screen "Prog_Lav2_1" 1366x768
   TextField "Campo de texto_1" at 49,16 size 194x39; Text 'LAVADORA 2'
   TextField "Campo de texto_2" at 49,80 size 103x23; Text 'ENJUAGUES'
   TextField "Campo de texto_3" at 49,112 size 90x23; Text 'INICIALES'
   TextField "Campo de texto_5" at 49,176 size 113x23; Text 'PRE-LAVADO'
   TextField "Campo de texto_10" at 49,336 size 88x23; Text 'LAVADO 1'
   TextField "Campo de texto_14" at 49,464 size 88x23; Text 'LAVADO 2'
   TextField "Campo de texto_18" at 49,592 size 103x23; Text 'ENJUAGUES'
   TextField "Campo de texto_19" at 49,624 size 74x23; Text 'FINALES'
   TextField "Campo de texto_20" at 49,656 size 137x23; Text 'CENTRIFUGADO'
   TextField "Campo de texto_27" at 193,80 size 94x23; Text 'CANTIDAD'
   TextField "Campo de texto_28" at 193,144 size 134x23; Text 'NIVEL DE AGUA'
   TextField "Campo de texto_29" at 193,112 size 70x23; Text 'TIEMPO'
   TextField "Campo de texto_30" at 193,208 size 134x23; Text 'NIVEL DE AGUA'
   TextField "Campo de texto_32" at 193,240 size 140x23; Text 'AGUA CALIENTE'
   TextField "Campo de texto_34" at 193,304 size 132x23; Text 'TEMPERATURA'
   TextField "Campo de texto_35" at 193,336 size 70x23; Text 'TIEMPO'
   TextField "Campo de texto_36" at 193,368 size 134x23; Text 'NIVEL DE AGUA'
   TextField "Campo de texto_37" at 193,400 size 140x23; Text 'AGUA CALIENTE'
   TextField "Campo de texto_38" at 193,432 size 132x23; Text 'TEMPERATURA'
   TextField "Campo de texto_39" at 193,464 size 70x23; Text 'TIEMPO'
   TextField "Campo de texto_40" at 193,496 size 134x23; Text 'NIVEL DE AGUA'
   TextField "Campo de texto_41" at 193,528 size 140x23; Text 'AGUA CALIENTE'
   TextField "Campo de texto_42" at 193,560 size 132x23; Text 'TEMPERATURA'
   TextField "Campo de texto_43" at 193,592 size 94x23; Text 'CANTIDAD'
   TextField "Campo de texto_44" at 193,624 size 70x23; Text 'TIEMPO'
   TextField "Campo de texto_45" at 193,656 size 70x23; Text 'TIEMPO'
   TextField "Campo de texto_4" at 193,272 size 63x23; Text 'VAPOR'
   TextField "Campo de texto_6" at 193,176 size 70x23; Text 'TIEMPO'
   TextField "Campo de texto_7" at 426,39 size 17x33; Text '9'
   TextField "Campo de texto_8" at 537,39 size 34x33; Text '10'
   TextField "Campo de texto_9" at 657,39 size 34x33; Text '11'
   TextField "Campo de texto_11" at 777,39 size 34x33; Text '12'
   TextField "Campo de texto_12" at 897,39 size 34x33; Text '13'
   TextField "Campo de texto_13" at 1017,39 size 34x33; Text '14'
   TextField "Campo de texto_15" at 1137,39 size 34x33; Text '15'
   TextField "Campo de texto_17" at 778,4 size 159x33; Text 'PROGRAMA'
   Button "Botón_1" at 6,695 size 361x66; TextOff 'ATRAS'
      on Click: ActivateScreen("Prog_Lav2_0", 0)
   Button "Botón_2" at 996,694 size 361x66; TextOff 'SIGUIENTE'
      on Click: ActivateScreen("Prog_Lav3_0", 0)
   Button "Botón_3" at 374,694 size 616x66; TextOff 'PRINCIPAL'
      on Click: ActivateScreen("Principal", 0)
   IOField "Campo ES_1" at 394,656 size 80x24; FormatPattern FF; Unit  M
      ProcessValue <- "Lav2_Prog9_Centr_Tiempo"
   IOField "Campo ES_2" at 394,592 size 80x24; FormatPattern F
      ProcessValue <- "Lav2_Prog9_EnjFin_Cant"
   IOField "Campo ES_3" at 394,624 size 80x24; FormatPattern FF; Unit  M
      ProcessValue <- "Lav2_Prog9_EnjFin_Tiempo"
   IOField "Campo ES_4" at 394,80 size 80x24; FormatPattern F
      ProcessValue <- "Lav2_Prog9_EnjIni_Cant"
   IOField "Campo ES_5" at 394,144 size 80x24; FormatPattern F
      ProcessValue <- "Lav2_Prog9_EnjIni_NivAg"
   IOField "Campo ES_6" at 394,112 size 80x24; FormatPattern FF; Unit  M
      ProcessValue <- "Lav2_Prog9_EnjIni_Tiempo"
   IOField "Campo ES_7" at 394,400 size 80x24; FormatPattern F
      ProcessValue <- "Lav2_Prog9_Lav1_AgCaliente"
   IOField "Campo ES_8" at 394,368 size 80x24; FormatPattern F
      ProcessValue <- "Lav2_Prog9_Lav1_NivAg"
   IOField "Campo ES_9" at 394,432 size 80x24; FormatPattern FF; Unit  °C
      ProcessValue <- "Lav2_Prog9_Lav1_Temperatura"
   IOField "Campo ES_10" at 394,336 size 80x24; FormatPattern FF; Unit  M
      ProcessValue <- "Lav2_Prog9_Lav1_Tiempo"
   IOField "Campo ES_11" at 394,528 size 80x24; FormatPattern F
      ProcessValue <- "Lav2_Prog9_Lav2_AgCaliente"
   IOField "Campo ES_12" at 394,496 size 80x24; FormatPattern F
      ProcessValue <- "Lav2_Prog9_Lav2_NivAg"
   IOField "Campo ES_13" at 394,560 size 80x24; FormatPattern FF; Unit °C
      ProcessValue <- "Lav2_Prog9_Lav2_Temperatura"
   IOField "Campo ES_14" at 394,464 size 80x24; FormatPattern FF; Unit  M
      ProcessValue <- "Lav2_Prog9_Lav2_Tiempo"
   IOField "Campo ES_15" at 394,240 size 80x24; FormatPattern F
      ProcessValue <- "Lav2_Prog9_PreLav_AgCaliente"
   IOField "Campo ES_16" at 394,208 size 80x24; FormatPattern F
      ProcessValue <- "Lav2_Prog9_PreLav_NivAg"
   IOField "Campo ES_17" at 394,304 size 80x24; FormatPattern FF; Unit  °C
      ProcessValue <- "Lav2_Prog9_PreLav_Temperatura"
   IOField "Campo ES_18" at 394,176 size 80x24; FormatPattern FF; Unit  M
      ProcessValue <- "Lav2_Prog9_PreLav_Tiempo"
   IOField "Campo ES_19" at 394,272 size 80x24; FormatPattern F
      ProcessValue <- "Lav2_Prog9_PreLav_Vapor"
   IOField "Campo ES_20" at 514,656 size 80x24; FormatPattern FF; Unit  M
      ProcessValue <- "Lav2_Prog10_Centr_Tiempo"
   IOField "Campo ES_21" at 514,592 size 80x24; FormatPattern F
      ProcessValue <- "Lav2_Prog10_EnjFin_Cant"
   IOField "Campo ES_22" at 514,624 size 80x24; FormatPattern FF; Unit  M
      ProcessValue <- "Lav2_Prog10_EnjFin_Tiempo"
   IOField "Campo ES_23" at 514,80 size 80x24; FormatPattern F
      ProcessValue <- "Lav2_Prog10_EnjIni_Cant"
   IOField "Campo ES_24" at 514,144 size 80x24; FormatPattern F
      ProcessValue <- "Lav2_Prog10_EnjIni_NivAg"
   IOField "Campo ES_25" at 514,112 size 80x24; FormatPattern FF; Unit  M
      ProcessValue <- "Lav2_Prog10_EnjIni_Tiempo"
   IOField "Campo ES_26" at 514,400 size 80x24; FormatPattern F
      ProcessValue <- "Lav2_Prog10_Lav1_AgCaliente"
   IOField "Campo ES_27" at 514,368 size 80x24; FormatPattern F
      ProcessValue <- "Lav2_Prog10_Lav1_NivAg"
   IOField "Campo ES_28" at 514,432 size 80x24; FormatPattern FF; Unit  °C
      ProcessValue <- "Lav2_Prog10_Lav1_Temperatura"
   IOField "Campo ES_29" at 514,336 size 80x24; FormatPattern FF; Unit  M
      ProcessValue <- "Lav2_Prog10_Lav1_Tiempo"
   IOField "Campo ES_30" at 514,528 size 80x24; FormatPattern F
      ProcessValue <- "Lav2_Prog10_Lav2_AgCaliente"
   IOField "Campo ES_31" at 514,496 size 80x24; FormatPattern F
      ProcessValue <- "Lav2_Prog10_Lav2_NivAg"
   IOField "Campo ES_32" at 514,560 size 80x24; FormatPattern FF; Unit °C
      ProcessValue <- "Lav2_Prog10_Lav2_Temperatura"
   IOField "Campo ES_33" at 514,464 size 80x24; FormatPattern FF; Unit  M
      ProcessValue <- "Lav2_Prog10_Lav2_Tiempo"
   IOField "Campo ES_34" at 514,240 size 80x24; FormatPattern F
      ProcessValue <- "Lav2_Prog10_PreLav_AgCaliente"
   IOField "Campo ES_35" at 514,208 size 80x24; FormatPattern F
      ProcessValue <- "Lav2_Prog10_PreLav_NivAg"
   IOField "Campo ES_36" at 514,304 size 80x24; FormatPattern FF; Unit  °C
      ProcessValue <- "Lav2_Prog10_PreLav_Temperatura"
   IOField "Campo ES_37" at 514,176 size 80x24; FormatPattern FF; Unit  M
      ProcessValue <- "Lav2_Prog10_PreLav_Tiempo"
   IOField "Campo ES_38" at 514,272 size 80x24; FormatPattern F
      ProcessValue <- "Lav2_Prog10_PreLav_Vapor"
   IOField "Campo ES_39" at 634,656 size 80x24; FormatPattern FF; Unit  M
      ProcessValue <- "Lav2_Prog11_Centr_Tiempo"
   IOField "Campo ES_40" at 634,592 size 80x24; FormatPattern F
      ProcessValue <- "Lav2_Prog11_EnjFin_Cant"
   IOField "Campo ES_41" at 634,624 size 80x24; FormatPattern FF; Unit  M
      ProcessValue <- "Lav2_Prog11_EnjFin_Tiempo"
   IOField "Campo ES_42" at 634,80 size 80x24; FormatPattern F
      ProcessValue <- "Lav2_Prog11_EnjIni_Cant"
   IOField "Campo ES_43" at 634,144 size 80x24; FormatPattern F
      ProcessValue <- "Lav2_Prog11_EnjIni_NivAg"
   IOField "Campo ES_44" at 634,112 size 80x24; FormatPattern FF; Unit  M
      ProcessValue <- "Lav2_Prog11_EnjIni_Tiempo"
   IOField "Campo ES_45" at 634,400 size 80x24; FormatPattern F
      ProcessValue <- "Lav2_Prog11_Lav1_AgCaliente"
   IOField "Campo ES_46" at 634,368 size 80x24; FormatPattern F
      ProcessValue <- "Lav2_Prog11_Lav1_NivAg"
   IOField "Campo ES_47" at 634,432 size 80x24; FormatPattern FF; Unit  °C
      ProcessValue <- "Lav2_Prog11_Lav1_Temperatura"
   IOField "Campo ES_48" at 634,336 size 80x24; FormatPattern FF; Unit  M
      ProcessValue <- "Lav2_Prog11_Lav1_Tiempo"
   IOField "Campo ES_49" at 634,528 size 80x24; FormatPattern F
      ProcessValue <- "Lav2_Prog11_Lav2_AgCaliente"
   IOField "Campo ES_50" at 634,496 size 80x24; FormatPattern F
      ProcessValue <- "Lav2_Prog11_Lav2_NivAg"
   IOField "Campo ES_51" at 634,560 size 80x24; FormatPattern FF; Unit °C
      ProcessValue <- "Lav2_Prog11_Lav2_Temperatura"
   IOField "Campo ES_52" at 634,464 size 80x24; FormatPattern FF; Unit  M
      ProcessValue <- "Lav2_Prog11_Lav2_Tiempo"
   IOField "Campo ES_53" at 634,240 size 80x24; FormatPattern F
      ProcessValue <- "Lav2_Prog11_PreLav_AgCaliente"
   IOField "Campo ES_54" at 634,208 size 80x24; FormatPattern F
      ProcessValue <- "Lav2_Prog11_PreLav_NivAg"
   IOField "Campo ES_55" at 634,304 size 80x24; FormatPattern FF; Unit  °C
      ProcessValue <- "Lav2_Prog11_PreLav_Temperatura"
   IOField "Campo ES_56" at 634,176 size 80x24; FormatPattern FF; Unit  M
      ProcessValue <- "Lav2_Prog11_PreLav_Tiempo"
   IOField "Campo ES_57" at 634,272 size 80x24; FormatPattern F
      ProcessValue <- "Lav2_Prog11_PreLav_Vapor"
   IOField "Campo ES_58" at 754,656 size 80x24; FormatPattern FF; Unit  M
      ProcessValue <- "Lav2_Prog12_Centr_Tiempo"
   IOField "Campo ES_59" at 754,592 size 80x24; FormatPattern F
      ProcessValue <- "Lav2_Prog12_EnjFin_Cant"
   IOField "Campo ES_60" at 754,624 size 80x24; FormatPattern FF; Unit  M
      ProcessValue <- "Lav2_Prog12_EnjFin_Tiempo"
   IOField "Campo ES_61" at 754,80 size 80x24; FormatPattern F
      ProcessValue <- "Lav2_Prog12_EnjIni_Cant"
   IOField "Campo ES_62" at 754,144 size 80x24; FormatPattern F
      ProcessValue <- "Lav2_Prog12_EnjIni_NivAg"
   IOField "Campo ES_63" at 754,112 size 80x24; FormatPattern FF; Unit  M
      ProcessValue <- "Lav2_Prog12_EnjIni_Tiempo"
   IOField "Campo ES_64" at 754,400 size 80x24; FormatPattern F
      ProcessValue <- "Lav2_Prog12_Lav1_AgCaliente"
   IOField "Campo ES_65" at 754,368 size 80x24; FormatPattern F
      ProcessValue <- "Lav2_Prog12_Lav1_NivAg"
   IOField "Campo ES_66" at 754,432 size 80x24; FormatPattern FF; Unit  °C
      ProcessValue <- "Lav2_Prog12_Lav1_Temperatura"
   IOField "Campo ES_67" at 754,336 size 80x24; FormatPattern FF; Unit  M
      ProcessValue <- "Lav2_Prog12_Lav1_Tiempo"
   IOField "Campo ES_68" at 754,528 size 80x24; FormatPattern F
      ProcessValue <- "Lav2_Prog12_Lav2_AgCaliente"
   IOField "Campo ES_69" at 754,496 size 80x24; FormatPattern F
      ProcessValue <- "Lav2_Prog12_Lav2_NivAg"
   IOField "Campo ES_70" at 754,560 size 80x24; FormatPattern FF; Unit °C
      ProcessValue <- "Lav2_Prog12_Lav2_Temperatura"
   IOField "Campo ES_71" at 754,464 size 80x24; FormatPattern FF; Unit  M
      ProcessValue <- "Lav2_Prog12_Lav2_Tiempo"
   IOField "Campo ES_72" at 754,240 size 80x24; FormatPattern F
      ProcessValue <- "Lav2_Prog12_PreLav_AgCaliente"
   IOField "Campo ES_73" at 754,208 size 80x24; FormatPattern F
      ProcessValue <- "Lav2_Prog12_PreLav_NivAg"
   IOField "Campo ES_74" at 754,304 size 80x24; FormatPattern FF; Unit  °C
      ProcessValue <- "Lav2_Prog12_PreLav_Temperatura"
   IOField "Campo ES_75" at 754,176 size 80x24; FormatPattern FF; Unit  M
      ProcessValue <- "Lav2_Prog12_PreLav_Tiempo"
   IOField "Campo ES_76" at 754,272 size 80x24; FormatPattern F
      ProcessValue <- "Lav2_Prog12_PreLav_Vapor"
   IOField "Campo ES_77" at 874,656 size 80x24; FormatPattern FF; Unit  M
      ProcessValue <- "Lav2_Prog13_Centr_Tiempo"
   IOField "Campo ES_78" at 874,592 size 80x24; FormatPattern F
      ProcessValue <- "Lav2_Prog13_EnjFin_Cant"
   IOField "Campo ES_79" at 874,624 size 80x24; FormatPattern FF; Unit  M
      ProcessValue <- "Lav2_Prog13_EnjFin_Tiempo"
   IOField "Campo ES_80" at 874,80 size 80x24; FormatPattern F
      ProcessValue <- "Lav2_Prog13_EnjIni_Cant"
   IOField "Campo ES_81" at 874,144 size 80x24; FormatPattern F
      ProcessValue <- "Lav2_Prog13_EnjIni_NivAg"
   IOField "Campo ES_82" at 874,112 size 80x24; FormatPattern FF; Unit  M
      ProcessValue <- "Lav2_Prog13_EnjIni_Tiempo"
   IOField "Campo ES_83" at 874,400 size 80x24; FormatPattern F
      ProcessValue <- "Lav2_Prog13_Lav1_AgCaliente"
   IOField "Campo ES_84" at 874,368 size 80x24; FormatPattern F
      ProcessValue <- "Lav2_Prog13_Lav1_NivAg"
   IOField "Campo ES_85" at 874,432 size 80x24; FormatPattern FF; Unit  °C
      ProcessValue <- "Lav2_Prog13_Lav1_Temperatura"
   IOField "Campo ES_86" at 874,336 size 80x24; FormatPattern FF; Unit  M
      ProcessValue <- "Lav2_Prog13_Lav1_Tiempo"
   IOField "Campo ES_87" at 874,528 size 80x24; FormatPattern F
      ProcessValue <- "Lav2_Prog13_Lav2_AgCaliente"
   IOField "Campo ES_88" at 874,496 size 80x24; FormatPattern F
      ProcessValue <- "Lav2_Prog13_Lav2_NivAg"
   IOField "Campo ES_89" at 874,560 size 80x24; FormatPattern FF; Unit °C
      ProcessValue <- "Lav2_Prog13_Lav2_Temperatura"
   IOField "Campo ES_90" at 874,464 size 80x24; FormatPattern FF; Unit  M
      ProcessValue <- "Lav2_Prog13_Lav2_Tiempo"
   IOField "Campo ES_91" at 874,240 size 80x24; FormatPattern F
      ProcessValue <- "Lav2_Prog13_PreLav_AgCaliente"
   IOField "Campo ES_92" at 874,208 size 80x24; FormatPattern F
      ProcessValue <- "Lav2_Prog13_PreLav_NivAg"
   IOField "Campo ES_93" at 874,304 size 80x24; FormatPattern FF; Unit  °C
      ProcessValue <- "Lav2_Prog13_PreLav_Temperatura"
   IOField "Campo ES_94" at 874,176 size 80x24; FormatPattern FF; Unit  M
      ProcessValue <- "Lav2_Prog13_PreLav_Tiempo"
   IOField "Campo ES_95" at 874,272 size 80x24; FormatPattern F
      ProcessValue <- "Lav2_Prog13_PreLav_Vapor"
   IOField "Campo ES_96" at 994,656 size 80x24; FormatPattern FF; Unit  M
      ProcessValue <- "Lav2_Prog14_Centr_Tiempo"
   IOField "Campo ES_97" at 994,592 size 80x24; FormatPattern F
      ProcessValue <- "Lav2_Prog14_EnjFin_Cant"
   IOField "Campo ES_98" at 994,624 size 80x24; FormatPattern FF; Unit  M
      ProcessValue <- "Lav2_Prog14_EnjFin_Tiempo"
   IOField "Campo ES_99" at 994,80 size 80x24; FormatPattern F
      ProcessValue <- "Lav2_Prog14_EnjIni_Cant"
   IOField "Campo ES_100" at 994,144 size 80x24; FormatPattern F
      ProcessValue <- "Lav2_Prog14_EnjIni_NivAg"
   IOField "Campo ES_101" at 994,112 size 80x24; FormatPattern FF; Unit  M
      ProcessValue <- "Lav2_Prog14_EnjIni_Tiempo"
   IOField "Campo ES_102" at 994,400 size 80x24; FormatPattern F
      ProcessValue <- "Lav2_Prog14_Lav1_AgCaliente"
   IOField "Campo ES_103" at 994,368 size 80x24; FormatPattern F
      ProcessValue <- "Lav2_Prog14_Lav1_NivAg"
   IOField "Campo ES_104" at 994,432 size 80x24; FormatPattern FF; Unit  °C
      ProcessValue <- "Lav2_Prog14_Lav1_Temperatura"
   IOField "Campo ES_105" at 994,336 size 80x24; FormatPattern FF; Unit  M
      ProcessValue <- "Lav2_Prog14_Lav1_Tiempo"
   IOField "Campo ES_106" at 994,528 size 80x24; FormatPattern F
      ProcessValue <- "Lav2_Prog14_Lav2_AgCaliente"
   IOField "Campo ES_107" at 994,496 size 80x24; FormatPattern F
      ProcessValue <- "Lav2_Prog14_Lav2_NivAg"
   IOField "Campo ES_108" at 994,560 size 80x24; FormatPattern FF; Unit °C
      ProcessValue <- "Lav2_Prog14_Lav2_Temperatura"
   IOField "Campo ES_109" at 994,464 size 80x24; FormatPattern FF; Unit  M
      ProcessValue <- "Lav2_Prog14_Lav2_Tiempo"
   IOField "Campo ES_110" at 994,240 size 80x24; FormatPattern F
      ProcessValue <- "Lav2_Prog14_PreLav_AgCaliente"
   IOField "Campo ES_111" at 994,208 size 80x24; FormatPattern F
      ProcessValue <- "Lav2_Prog14_PreLav_NivAg"
   IOField "Campo ES_112" at 994,304 size 80x24; FormatPattern FF; Unit  °C
      ProcessValue <- "Lav2_Prog14_PreLav_Temperatura"
   IOField "Campo ES_113" at 994,176 size 80x24; FormatPattern FF; Unit  M
      ProcessValue <- "Lav2_Prog14_PreLav_Tiempo"
   IOField "Campo ES_114" at 994,272 size 80x24; FormatPattern F
      ProcessValue <- "Lav2_Prog14_PreLav_Vapor"
   IOField "Campo ES_115" at 1114,656 size 80x24; FormatPattern FF; Unit  M
      ProcessValue <- "Lav2_Prog15_Centr_Tiempo"
   IOField "Campo ES_116" at 1114,592 size 80x24; FormatPattern F
      ProcessValue <- "Lav2_Prog15_EnjFin_Cant"
   IOField "Campo ES_117" at 1114,624 size 80x24; FormatPattern FF; Unit  M
      ProcessValue <- "Lav2_Prog15_EnjFin_Tiempo"
   IOField "Campo ES_118" at 1114,80 size 80x24; FormatPattern F
      ProcessValue <- "Lav2_Prog15_EnjIni_Cant"
   IOField "Campo ES_119" at 1114,144 size 80x24; FormatPattern F
      ProcessValue <- "Lav2_Prog15_EnjIni_NivAg"
   IOField "Campo ES_120" at 1114,112 size 80x24; FormatPattern FF; Unit  M
      ProcessValue <- "Lav2_Prog15_EnjIni_Tiempo"
   IOField "Campo ES_121" at 1114,400 size 80x24; FormatPattern F
      ProcessValue <- "Lav2_Prog15_Lav1_AgCaliente"
   IOField "Campo ES_122" at 1114,368 size 80x24; FormatPattern F
      ProcessValue <- "Lav2_Prog15_Lav1_NivAg"
   IOField "Campo ES_123" at 1114,432 size 80x24; FormatPattern FF; Unit  °C
      ProcessValue <- "Lav2_Prog15_Lav1_Temperatura"
   IOField "Campo ES_124" at 1114,336 size 80x24; FormatPattern FF; Unit  M
      ProcessValue <- "Lav2_Prog15_Lav1_Tiempo"
   IOField "Campo ES_125" at 1114,528 size 80x24; FormatPattern F
      ProcessValue <- "Lav2_Prog15_Lav2_AgCaliente"
   IOField "Campo ES_126" at 1114,496 size 80x24; FormatPattern F
      ProcessValue <- "Lav2_Prog15_Lav2_NivAg"
   IOField "Campo ES_127" at 1114,560 size 80x24; FormatPattern FF; Unit °C
      ProcessValue <- "Lav2_Prog15_Lav2_Temperatura"
   IOField "Campo ES_128" at 1114,464 size 80x24; FormatPattern FF; Unit  M
      ProcessValue <- "Lav2_Prog15_Lav2_Tiempo"
   IOField "Campo ES_129" at 1114,240 size 80x24; FormatPattern F
      ProcessValue <- "Lav2_Prog15_PreLav_AgCaliente"
   IOField "Campo ES_130" at 1114,208 size 80x24; FormatPattern F
      ProcessValue <- "Lav2_Prog15_PreLav_NivAg"
   IOField "Campo ES_131" at 1114,304 size 80x24; FormatPattern FF; Unit  °C
      ProcessValue <- "Lav2_Prog15_PreLav_Temperatura"
   IOField "Campo ES_132" at 1114,176 size 80x24; FormatPattern FF; Unit  M
      ProcessValue <- "Lav2_Prog15_PreLav_Tiempo"
   IOField "Campo ES_133" at 1114,272 size 80x24; FormatPattern F
      ProcessValue <- "Lav2_Prog15_PreLav_Vapor"

screen "Prog_Lav3_0" 1366x768
   TextField "Campo de texto_1" at 49,16 size 194x39; Text 'LAVADORA 3'
   TextField "Campo de texto_2" at 49,80 size 103x23; Text 'ENJUAGUES'
   TextField "Campo de texto_3" at 49,112 size 90x23; Text 'INICIALES'
   TextField "Campo de texto_5" at 49,176 size 113x23; Text 'PRE-LAVADO'
   TextField "Campo de texto_10" at 49,336 size 88x23; Text 'LAVADO 1'
   TextField "Campo de texto_14" at 49,464 size 88x23; Text 'LAVADO 2'
   TextField "Campo de texto_18" at 49,592 size 103x23; Text 'ENJUAGUES'
   TextField "Campo de texto_19" at 49,624 size 74x23; Text 'FINALES'
   TextField "Campo de texto_20" at 49,656 size 137x23; Text 'CENTRIFUGADO'
   TextField "Campo de texto_27" at 193,80 size 94x23; Text 'CANTIDAD'
   TextField "Campo de texto_28" at 193,144 size 134x23; Text 'NIVEL DE AGUA'
   TextField "Campo de texto_29" at 193,112 size 70x23; Text 'TIEMPO'
   TextField "Campo de texto_30" at 193,208 size 134x23; Text 'NIVEL DE AGUA'
   TextField "Campo de texto_32" at 193,240 size 140x23; Text 'AGUA CALIENTE'
   TextField "Campo de texto_34" at 193,304 size 132x23; Text 'TEMPERATURA'
   TextField "Campo de texto_35" at 193,336 size 70x23; Text 'TIEMPO'
   TextField "Campo de texto_36" at 193,368 size 134x23; Text 'NIVEL DE AGUA'
   TextField "Campo de texto_37" at 193,400 size 140x23; Text 'AGUA CALIENTE'
   TextField "Campo de texto_38" at 193,432 size 132x23; Text 'TEMPERATURA'
   TextField "Campo de texto_39" at 193,464 size 70x23; Text 'TIEMPO'
   TextField "Campo de texto_40" at 193,496 size 134x23; Text 'NIVEL DE AGUA'
   TextField "Campo de texto_41" at 193,528 size 140x23; Text 'AGUA CALIENTE'
   TextField "Campo de texto_42" at 193,560 size 132x23; Text 'TEMPERATURA'
   TextField "Campo de texto_43" at 193,592 size 94x23; Text 'CANTIDAD'
   TextField "Campo de texto_44" at 193,624 size 70x23; Text 'TIEMPO'
   TextField "Campo de texto_45" at 193,656 size 70x23; Text 'TIEMPO'
   TextField "Campo de texto_4" at 193,272 size 63x23; Text 'VAPOR'
   TextField "Campo de texto_6" at 193,176 size 70x23; Text 'TIEMPO'
   TextField "Campo de texto_7" at 426,39 size 17x33; Text '1'
   TextField "Campo de texto_8" at 546,39 size 17x33; Text '2'
   TextField "Campo de texto_9" at 666,39 size 17x33; Text '3'
   TextField "Campo de texto_11" at 786,39 size 17x33; Text '4'
   TextField "Campo de texto_12" at 906,39 size 17x33; Text '5'
   TextField "Campo de texto_13" at 1026,39 size 17x33; Text '6'
   TextField "Campo de texto_15" at 1146,39 size 17x33; Text '7'
   TextField "Campo de texto_16" at 1266,39 size 17x33; Text '8'
   TextField "Campo de texto_17" at 778,4 size 159x33; Text 'PROGRAMA'
   Button "Botón_1" at 6,695 size 361x66; TextOff 'ATRAS'
      on Click: ActivateScreen("Prog_Lav2_1", 0)
   Button "Botón_2" at 996,694 size 361x66; TextOff 'SIGUIENTE'
      on Click: ActivateScreen("Prog_Lav3_1", 0)
   Button "Botón_3" at 374,694 size 616x66; TextOff 'PRINCIPAL'
      on Click: ActivateScreen("Principal", 0)
   IOField "Campo ES_1" at 394,656 size 80x24; FormatPattern FF; Unit  M
      ProcessValue <- "Lav3_Prog1_Centr_Tiempo"
   IOField "Campo ES_2" at 394,592 size 80x24; FormatPattern F
      ProcessValue <- "Lav3_Prog1_EnjFin_Cant"
   IOField "Campo ES_3" at 394,624 size 80x24; FormatPattern FF; Unit  M
      ProcessValue <- "Lav3_Prog1_EnjFin_Tiempo"
   IOField "Campo ES_4" at 394,80 size 80x24; FormatPattern F
      ProcessValue <- "Lav3_Prog1_EnjIni_Cant"
   IOField "Campo ES_5" at 394,144 size 80x24; FormatPattern F
      ProcessValue <- "Lav3_Prog1_EnjIni_NivAg"
   IOField "Campo ES_6" at 394,112 size 80x24; FormatPattern FF; Unit  M
      ProcessValue <- "Lav3_Prog1_EnjIni_Tiempo"
   IOField "Campo ES_7" at 394,400 size 80x24; FormatPattern F
      ProcessValue <- "Lav3_Prog1_Lav1_AgCaliente"
   IOField "Campo ES_8" at 394,368 size 80x24; FormatPattern F
      ProcessValue <- "Lav3_Prog1_Lav1_NivAg"
   IOField "Campo ES_9" at 394,432 size 80x24; FormatPattern FF; Unit  °C
      ProcessValue <- "Lav3_Prog1_Lav1_Temperatura"
   IOField "Campo ES_10" at 394,336 size 80x24; FormatPattern FF; Unit  M
      ProcessValue <- "Lav3_Prog1_Lav1_Tiempo"
   IOField "Campo ES_11" at 394,528 size 80x24; FormatPattern F
      ProcessValue <- "Lav3_Prog1_Lav2_AgCaliente"
   IOField "Campo ES_12" at 394,496 size 80x24; FormatPattern F
      ProcessValue <- "Lav3_Prog1_Lav2_NivAg"
   IOField "Campo ES_13" at 394,560 size 80x24; FormatPattern FF; Unit °C
      ProcessValue <- "Lav3_Prog1_Lav2_Temperatura"
   IOField "Campo ES_14" at 394,464 size 80x24; FormatPattern FF; Unit  M
      ProcessValue <- "Lav3_Prog1_Lav2_Tiempo"
   IOField "Campo ES_15" at 394,240 size 80x24; FormatPattern F
      ProcessValue <- "Lav3_Prog1_PreLav_AgCaliente"
   IOField "Campo ES_16" at 394,208 size 80x24; FormatPattern F
      ProcessValue <- "Lav3_Prog1_PreLav_NivAg"
   IOField "Campo ES_17" at 394,304 size 80x24; FormatPattern FF; Unit  °C
      ProcessValue <- "Lav3_Prog1_PreLav_Temperatura"
   IOField "Campo ES_18" at 394,176 size 80x24; FormatPattern FF; Unit  M
      ProcessValue <- "Lav3_Prog1_PreLav_Tiempo"
   IOField "Campo ES_19" at 394,272 size 80x24; FormatPattern F
      ProcessValue <- "Lav3_Prog1_PreLav_Vapor"
   IOField "Campo ES_20" at 514,656 size 80x24; FormatPattern FF; Unit  M
      ProcessValue <- "Lav3_Prog2_Centr_Tiempo"
   IOField "Campo ES_21" at 514,592 size 80x24; FormatPattern F
      ProcessValue <- "Lav3_Prog2_EnjFin_Cant"
   IOField "Campo ES_22" at 514,624 size 80x24; FormatPattern FF; Unit  M
      ProcessValue <- "Lav3_Prog2_EnjFin_Tiempo"
   IOField "Campo ES_23" at 514,80 size 80x24; FormatPattern F
      ProcessValue <- "Lav3_Prog2_EnjIni_Cant"
   IOField "Campo ES_24" at 514,144 size 80x24; FormatPattern F
      ProcessValue <- "Lav3_Prog2_EnjIni_NivAg"
   IOField "Campo ES_25" at 514,112 size 80x24; FormatPattern FF; Unit  M
      ProcessValue <- "Lav3_Prog2_EnjIni_Tiempo"
   IOField "Campo ES_26" at 514,400 size 80x24; FormatPattern F
      ProcessValue <- "Lav3_Prog2_Lav1_AgCaliente"
   IOField "Campo ES_27" at 514,368 size 80x24; FormatPattern F
      ProcessValue <- "Lav3_Prog2_Lav1_NivAg"
   IOField "Campo ES_28" at 514,432 size 80x24; FormatPattern FF; Unit  °C
      ProcessValue <- "Lav3_Prog2_Lav1_Temperatura"
   IOField "Campo ES_29" at 514,336 size 80x24; FormatPattern FF; Unit  M
      ProcessValue <- "Lav3_Prog2_Lav1_Tiempo"
   IOField "Campo ES_30" at 514,528 size 80x24; FormatPattern F
      ProcessValue <- "Lav3_Prog2_Lav2_AgCaliente"
   IOField "Campo ES_31" at 514,496 size 80x24; FormatPattern F
      ProcessValue <- "Lav3_Prog2_Lav2_NivAg"
   IOField "Campo ES_32" at 514,560 size 80x24; FormatPattern FF; Unit °C
      ProcessValue <- "Lav3_Prog2_Lav2_Temperatura"
   IOField "Campo ES_33" at 514,464 size 80x24; FormatPattern FF; Unit  M
      ProcessValue <- "Lav3_Prog2_Lav2_Tiempo"
   IOField "Campo ES_34" at 514,240 size 80x24; FormatPattern F
      ProcessValue <- "Lav3_Prog2_PreLav_AgCaliente"
   IOField "Campo ES_35" at 514,208 size 80x24; FormatPattern F
      ProcessValue <- "Lav3_Prog2_PreLav_NivAg"
   IOField "Campo ES_36" at 514,304 size 80x24; FormatPattern FF; Unit  °C
      ProcessValue <- "Lav3_Prog2_PreLav_Temperatura"
   IOField "Campo ES_37" at 514,176 size 80x24; FormatPattern FF; Unit  M
      ProcessValue <- "Lav3_Prog2_PreLav_Tiempo"
   IOField "Campo ES_38" at 514,272 size 80x24; FormatPattern F
      ProcessValue <- "Lav3_Prog2_PreLav_Vapor"
   IOField "Campo ES_39" at 634,656 size 80x24; FormatPattern FF; Unit  M
      ProcessValue <- "Lav3_Prog3_Centr_Tiempo"
   IOField "Campo ES_40" at 634,592 size 80x24; FormatPattern F
      ProcessValue <- "Lav3_Prog3_EnjFin_Cant"
   IOField "Campo ES_41" at 634,624 size 80x24; FormatPattern FF; Unit  M
      ProcessValue <- "Lav3_Prog3_EnjFin_Tiempo"
   IOField "Campo ES_42" at 634,80 size 80x24; FormatPattern F
      ProcessValue <- "Lav3_Prog3_EnjIni_Cant"
   IOField "Campo ES_43" at 634,144 size 80x24; FormatPattern F
      ProcessValue <- "Lav3_Prog3_EnjIni_NivAg"
   IOField "Campo ES_44" at 634,112 size 80x24; FormatPattern FF; Unit  M
      ProcessValue <- "Lav3_Prog3_EnjIni_Tiempo"
   IOField "Campo ES_45" at 634,400 size 80x24; FormatPattern F
      ProcessValue <- "Lav3_Prog3_Lav1_AgCaliente"
   IOField "Campo ES_46" at 634,368 size 80x24; FormatPattern F
      ProcessValue <- "Lav3_Prog3_Lav1_NivAg"
   IOField "Campo ES_47" at 634,432 size 80x24; FormatPattern FF; Unit  °C
      ProcessValue <- "Lav3_Prog3_Lav1_Temperatura"
   IOField "Campo ES_48" at 634,336 size 80x24; FormatPattern FF; Unit  M
      ProcessValue <- "Lav3_Prog3_Lav1_Tiempo"
   IOField "Campo ES_49" at 634,528 size 80x24; FormatPattern F
      ProcessValue <- "Lav3_Prog3_Lav2_AgCaliente"
   IOField "Campo ES_50" at 634,496 size 80x24; FormatPattern F
      ProcessValue <- "Lav3_Prog3_Lav2_NivAg"
   IOField "Campo ES_51" at 634,560 size 80x24; FormatPattern FF; Unit °C
      ProcessValue <- "Lav3_Prog3_Lav2_Temperatura"
   IOField "Campo ES_52" at 634,464 size 80x24; FormatPattern FF; Unit  M
      ProcessValue <- "Lav3_Prog3_Lav2_Tiempo"
   IOField "Campo ES_53" at 634,240 size 80x24; FormatPattern F
      ProcessValue <- "Lav3_Prog3_PreLav_AgCaliente"
   IOField "Campo ES_54" at 634,208 size 80x24; FormatPattern F
      ProcessValue <- "Lav3_Prog3_PreLav_NivAg"
   IOField "Campo ES_55" at 634,304 size 80x24; FormatPattern FF; Unit  °C
      ProcessValue <- "Lav3_Prog3_PreLav_Temperatura"
   IOField "Campo ES_56" at 634,176 size 80x24; FormatPattern FF; Unit  M
      ProcessValue <- "Lav3_Prog3_PreLav_Tiempo"
   IOField "Campo ES_57" at 634,272 size 80x24; FormatPattern F
      ProcessValue <- "Lav3_Prog3_PreLav_Vapor"
   IOField "Campo ES_58" at 754,656 size 80x24; FormatPattern FF; Unit  M
      ProcessValue <- "Lav3_Prog4_Centr_Tiempo"
   IOField "Campo ES_59" at 754,592 size 80x24; FormatPattern F
      ProcessValue <- "Lav1_Prog4_EnjFin_Cant"
   IOField "Campo ES_60" at 754,624 size 80x24; FormatPattern FF; Unit  M
      ProcessValue <- "Lav1_Prog4_EnjFin_Tiempo"
   IOField "Campo ES_61" at 754,80 size 80x24; FormatPattern F
      ProcessValue <- "Lav1_Prog4_EnjIni_Cant"
   IOField "Campo ES_62" at 754,144 size 80x24; FormatPattern F
      ProcessValue <- "Lav1_Prog4_EnjIni_NivAg"
   IOField "Campo ES_63" at 754,112 size 80x24; FormatPattern FF; Unit  M
      ProcessValue <- "Lav1_Prog4_EnjIni_Tiempo"
   IOField "Campo ES_64" at 754,400 size 80x24; FormatPattern F
      ProcessValue <- "Lav1_Prog4_Lav1_AgCaliente"
   IOField "Campo ES_65" at 754,368 size 80x24; FormatPattern F
      ProcessValue <- "Lav1_Prog4_Lav1_NivAg"
   IOField "Campo ES_66" at 754,432 size 80x24; FormatPattern FF; Unit  °C
      ProcessValue <- "Lav1_Prog4_Lav1_Temperatura"
   IOField "Campo ES_67" at 754,336 size 80x24; FormatPattern FF; Unit  M
      ProcessValue <- "Lav1_Prog4_Lav1_Tiempo"
   IOField "Campo ES_68" at 754,528 size 80x24; FormatPattern F
      ProcessValue <- "Lav1_Prog4_Lav2_AgCaliente"
   IOField "Campo ES_69" at 754,496 size 80x24; FormatPattern F
      ProcessValue <- "Lav1_Prog4_Lav2_NivAg"
   IOField "Campo ES_70" at 754,560 size 80x24; FormatPattern FF; Unit °C
      ProcessValue <- "Lav1_Prog4_Lav2_Temperatura"
   IOField "Campo ES_71" at 754,464 size 80x24; FormatPattern FF; Unit  M
      ProcessValue <- "Lav1_Prog4_Lav2_Tiempo"
   IOField "Campo ES_72" at 754,240 size 80x24; FormatPattern F
      ProcessValue <- "Lav1_Prog4_PreLav_AgCaliente"
   IOField "Campo ES_73" at 754,208 size 80x24; FormatPattern F
      ProcessValue <- "Lav1_Prog4_PreLav_NivAg"
   IOField "Campo ES_74" at 754,304 size 80x24; FormatPattern FF; Unit  °C
      ProcessValue <- "Lav1_Prog4_PreLav_Temperatura"
   IOField "Campo ES_75" at 754,176 size 80x24; FormatPattern FF; Unit  M
      ProcessValue <- "Lav1_Prog4_PreLav_Tiempo"
   IOField "Campo ES_76" at 754,272 size 80x24; FormatPattern F
      ProcessValue <- "Lav1_Prog4_PreLav_Vapor"
   IOField "Campo ES_77" at 874,656 size 80x24; FormatPattern FF; Unit  M
      ProcessValue <- "Lav3_Prog6_Centr_Tiempo"
   IOField "Campo ES_78" at 874,592 size 80x24; FormatPattern F
      ProcessValue <- "Lav3_Prog6_EnjFin_Cant"
   IOField "Campo ES_79" at 874,624 size 80x24; FormatPattern FF; Unit  M
      ProcessValue <- "Lav3_Prog6_EnjFin_Tiempo"
   IOField "Campo ES_80" at 874,80 size 80x24; FormatPattern F
      ProcessValue <- "Lav3_Prog5_EnjIni_Cant"
   IOField "Campo ES_81" at 874,144 size 80x24; FormatPattern F
      ProcessValue <- "Lav3_Prog5_EnjIni_NivAg"
   IOField "Campo ES_82" at 874,112 size 80x24; FormatPattern FF; Unit  M
      ProcessValue <- "Lav3_Prog5_EnjIni_Tiempo"
   IOField "Campo ES_83" at 874,400 size 80x24; FormatPattern F
      ProcessValue <- "Lav3_Prog5_Lav1_AgCaliente"
   IOField "Campo ES_84" at 874,368 size 80x24; FormatPattern F
      ProcessValue <- "Lav3_Prog5_Lav1_NivAg"
   IOField "Campo ES_85" at 874,432 size 80x24; FormatPattern FF; Unit  °C
      ProcessValue <- "Lav3_Prog5_Lav1_Temperatura"
   IOField "Campo ES_86" at 874,336 size 80x24; FormatPattern FF; Unit  M
      ProcessValue <- "Lav3_Prog5_Lav1_Tiempo"
   IOField "Campo ES_87" at 874,528 size 80x24; FormatPattern F
      ProcessValue <- "Lav3_Prog6_Lav2_AgCaliente"
   IOField "Campo ES_88" at 874,496 size 80x24; FormatPattern F
      ProcessValue <- "Lav3_Prog6_Lav2_NivAg"
   IOField "Campo ES_89" at 874,560 size 80x24; FormatPattern FF; Unit °C
      ProcessValue <- "Lav3_Prog6_Lav2_Temperatura"
   IOField "Campo ES_90" at 874,464 size 80x24; FormatPattern FF; Unit  M
      ProcessValue <- "Lav3_Prog6_Lav2_Tiempo"
   IOField "Campo ES_91" at 874,240 size 80x24; FormatPattern F
      ProcessValue <- "Lav3_Prog5_PreLav_AgCaliente"
   IOField "Campo ES_92" at 874,208 size 80x24; FormatPattern F
      ProcessValue <- "Lav3_Prog5_PreLav_NivAg"
   IOField "Campo ES_93" at 874,304 size 80x24; FormatPattern FF; Unit  °C
      ProcessValue <- "Lav3_Prog5_PreLav_Temperatura"
   IOField "Campo ES_94" at 874,176 size 80x24; FormatPattern FF; Unit  M
      ProcessValue <- "Lav3_Prog5_PreLav_Tiempo"
   IOField "Campo ES_95" at 874,272 size 80x24; FormatPattern F
      ProcessValue <- "Lav3_Prog5_PreLav_Vapor"
   IOField "Campo ES_96" at 994,656 size 80x24; FormatPattern FF; Unit  M
      ProcessValue <- "Lav3_Prog6_Centr_Tiempo"
   IOField "Campo ES_97" at 994,592 size 80x24; FormatPattern F
      ProcessValue <- "Lav3_Prog6_EnjFin_Cant"
   IOField "Campo ES_98" at 994,624 size 80x24; FormatPattern FF; Unit  M
      ProcessValue <- "Lav3_Prog6_EnjFin_Tiempo"
   IOField "Campo ES_99" at 994,80 size 80x24; FormatPattern F
      ProcessValue <- "Lav3_Prog6_EnjIni_Cant"
   IOField "Campo ES_100" at 994,144 size 80x24; FormatPattern F
      ProcessValue <- "Lav3_Prog6_EnjIni_NivAg"
   IOField "Campo ES_101" at 994,112 size 80x24; FormatPattern FF; Unit  M
      ProcessValue <- "Lav3_Prog6_EnjIni_Tiempo"
   IOField "Campo ES_102" at 994,400 size 80x24; FormatPattern F
      ProcessValue <- "Lav3_Prog6_Lav1_AgCaliente"
   IOField "Campo ES_103" at 994,368 size 80x24; FormatPattern F
      ProcessValue <- "Lav3_Prog6_Lav1_NivAg"
   IOField "Campo ES_104" at 994,432 size 80x24; FormatPattern FF; Unit  °C
      ProcessValue <- "Lav3_Prog6_Lav1_Temperatura"
   IOField "Campo ES_105" at 994,336 size 80x24; FormatPattern FF; Unit  M
      ProcessValue <- "Lav3_Prog6_Lav1_Tiempo"
   IOField "Campo ES_106" at 994,528 size 80x24; FormatPattern F
      ProcessValue <- "Lav3_Prog6_Lav2_AgCaliente"
   IOField "Campo ES_107" at 994,496 size 80x24; FormatPattern F
      ProcessValue <- "Lav3_Prog6_Lav2_NivAg"
   IOField "Campo ES_108" at 994,560 size 80x24; FormatPattern FF; Unit °C
      ProcessValue <- "Lav3_Prog6_Lav2_Temperatura"
   IOField "Campo ES_109" at 994,464 size 80x24; FormatPattern FF; Unit  M
      ProcessValue <- "Lav3_Prog6_Lav2_Tiempo"
   IOField "Campo ES_110" at 994,240 size 80x24; FormatPattern F
      ProcessValue <- "Lav3_Prog6_PreLav_AgCaliente"
   IOField "Campo ES_111" at 994,208 size 80x24; FormatPattern F
      ProcessValue <- "Lav3_Prog6_PreLav_NivAg"
   IOField "Campo ES_112" at 994,304 size 80x24; FormatPattern FF; Unit  °C
      ProcessValue <- "Lav3_Prog6_PreLav_Temperatura"
   IOField "Campo ES_113" at 994,176 size 80x24; FormatPattern FF; Unit  M
      ProcessValue <- "Lav3_Prog6_PreLav_Tiempo"
   IOField "Campo ES_114" at 994,272 size 80x24; FormatPattern F
      ProcessValue <- "Lav3_Prog6_PreLav_Vapor"
   IOField "Campo ES_115" at 1114,656 size 80x24; FormatPattern FF; Unit  M
      ProcessValue <- "Lav3_Prog7_Centr_Tiempo"
   IOField "Campo ES_116" at 1114,592 size 80x24; FormatPattern F
      ProcessValue <- "Lav3_Prog7_EnjFin_Cant"
   IOField "Campo ES_117" at 1114,624 size 80x24; FormatPattern FF; Unit  M
      ProcessValue <- "Lav3_Prog7_EnjFin_Tiempo"
   IOField "Campo ES_118" at 1114,80 size 80x24; FormatPattern F
      ProcessValue <- "Lav3_Prog7_EnjIni_Cant"
   IOField "Campo ES_119" at 1114,144 size 80x24; FormatPattern F
      ProcessValue <- "Lav3_Prog7_EnjIni_NivAg"
   IOField "Campo ES_120" at 1114,112 size 80x24; FormatPattern FF; Unit  M
      ProcessValue <- "Lav3_Prog7_EnjIni_Tiempo"
   IOField "Campo ES_121" at 1114,400 size 80x24; FormatPattern F
      ProcessValue <- "Lav3_Prog7_Lav1_AgCaliente"
   IOField "Campo ES_122" at 1114,368 size 80x24; FormatPattern F
      ProcessValue <- "Lav3_Prog7_Lav1_NivAg"
   IOField "Campo ES_123" at 1114,432 size 80x24; FormatPattern FF; Unit  °C
      ProcessValue <- "Lav3_Prog7_Lav1_Temperatura"
   IOField "Campo ES_124" at 1114,336 size 80x24; FormatPattern FF; Unit  M
      ProcessValue <- "Lav3_Prog7_Lav1_Tiempo"
   IOField "Campo ES_125" at 1114,528 size 80x24; FormatPattern F
      ProcessValue <- "Lav3_Prog7_Lav2_AgCaliente"
   IOField "Campo ES_126" at 1114,496 size 80x24; FormatPattern F
      ProcessValue <- "Lav3_Prog7_Lav2_NivAg"
   IOField "Campo ES_127" at 1114,560 size 80x24; FormatPattern FF; Unit °C
      ProcessValue <- "Lav3_Prog7_Lav2_Temperatura"
   IOField "Campo ES_128" at 1114,464 size 80x24; FormatPattern FF; Unit  M
      ProcessValue <- "Lav3_Prog7_Lav2_Tiempo"
   IOField "Campo ES_129" at 1114,240 size 80x24; FormatPattern F
      ProcessValue <- "Lav3_Prog7_PreLav_AgCaliente"
   IOField "Campo ES_130" at 1114,208 size 80x24; FormatPattern F
      ProcessValue <- "Lav3_Prog7_PreLav_NivAg"
   IOField "Campo ES_131" at 1114,304 size 80x24; FormatPattern FF; Unit  °C
      ProcessValue <- "Lav3_Prog7_PreLav_Temperatura"
   IOField "Campo ES_132" at 1114,176 size 80x24; FormatPattern FF; Unit  M
      ProcessValue <- "Lav3_Prog7_PreLav_Tiempo"
   IOField "Campo ES_133" at 1114,272 size 80x24; FormatPattern F
      ProcessValue <- "Lav3_Prog7_PreLav_Vapor"
   IOField "Campo ES_134" at 1234,656 size 80x24; FormatPattern FF; Unit  M
      ProcessValue <- "Lav3_Prog8_Centr_Tiempo"
   IOField "Campo ES_135" at 1234,592 size 80x24; FormatPattern F
      ProcessValue <- "Lav3_Prog8_EnjFin_Cant"
   IOField "Campo ES_136" at 1234,624 size 80x24; FormatPattern FF; Unit  M
      ProcessValue <- "Lav3_Prog8_EnjFin_Tiempo"
   IOField "Campo ES_137" at 1234,80 size 80x24; FormatPattern F
      ProcessValue <- "Lav3_Prog8_EnjIni_Cant"
   IOField "Campo ES_138" at 1234,144 size 80x24; FormatPattern F
      ProcessValue <- "Lav3_Prog8_EnjIni_NivAg"
   IOField "Campo ES_139" at 1234,112 size 80x24; FormatPattern FF; Unit  M
      ProcessValue <- "Lav3_Prog8_EnjIni_Tiempo"
   IOField "Campo ES_140" at 1234,400 size 80x24; FormatPattern F
      ProcessValue <- "Lav3_Prog8_Lav1_AgCaliente"
   IOField "Campo ES_141" at 1234,368 size 80x24; FormatPattern F
      ProcessValue <- "Lav3_Prog8_Lav1_NivAg"
   IOField "Campo ES_142" at 1234,432 size 80x24; FormatPattern FF; Unit  °C
      ProcessValue <- "Lav3_Prog8_Lav1_Temperatura"
   IOField "Campo ES_143" at 1234,336 size 80x24; FormatPattern FF; Unit  M
      ProcessValue <- "Lav3_Prog8_Lav1_Tiempo"
   IOField "Campo ES_144" at 1234,528 size 80x24; FormatPattern F
      ProcessValue <- "Lav3_Prog8_Lav2_AgCaliente"
   IOField "Campo ES_145" at 1234,496 size 80x24; FormatPattern F
      ProcessValue <- "Lav3_Prog8_Lav2_NivAg"
   IOField "Campo ES_146" at 1234,560 size 80x24; FormatPattern FF; Unit °C
      ProcessValue <- "Lav3_Prog8_Lav2_Temperatura"
   IOField "Campo ES_147" at 1234,464 size 80x24; FormatPattern FF; Unit  M
      ProcessValue <- "Lav3_Prog8_Lav2_Tiempo"
   IOField "Campo ES_148" at 1234,240 size 80x24; FormatPattern F
      ProcessValue <- "Lav3_Prog8_PreLav_AgCaliente"
   IOField "Campo ES_149" at 1234,208 size 80x24; FormatPattern F
      ProcessValue <- "Lav3_Prog8_PreLav_NivAg"
   IOField "Campo ES_150" at 1234,304 size 80x24; FormatPattern FF; Unit  °C
      ProcessValue <- "Lav3_Prog8_PreLav_Temperatura"
   IOField "Campo ES_151" at 1234,176 size 80x24; FormatPattern FF; Unit  M
      ProcessValue <- "Lav3_Prog8_PreLav_Tiempo"
   IOField "Campo ES_152" at 1234,272 size 80x24; FormatPattern F
      ProcessValue <- "Lav3_Prog8_PreLav_Vapor"

screen "Prog_Lav3_1" 1366x768
   TextField "Campo de texto_1" at 49,16 size 194x39; Text 'LAVADORA 3'
   TextField "Campo de texto_2" at 49,80 size 103x23; Text 'ENJUAGUES'
   TextField "Campo de texto_3" at 49,112 size 90x23; Text 'INICIALES'
   TextField "Campo de texto_5" at 49,176 size 113x23; Text 'PRE-LAVADO'
   TextField "Campo de texto_10" at 49,336 size 88x23; Text 'LAVADO 1'
   TextField "Campo de texto_14" at 49,464 size 88x23; Text 'LAVADO 2'
   TextField "Campo de texto_18" at 49,592 size 103x23; Text 'ENJUAGUES'
   TextField "Campo de texto_19" at 49,624 size 74x23; Text 'FINALES'
   TextField "Campo de texto_20" at 49,656 size 137x23; Text 'CENTRIFUGADO'
   TextField "Campo de texto_27" at 193,80 size 94x23; Text 'CANTIDAD'
   TextField "Campo de texto_28" at 193,144 size 134x23; Text 'NIVEL DE AGUA'
   TextField "Campo de texto_29" at 193,112 size 70x23; Text 'TIEMPO'
   TextField "Campo de texto_30" at 193,208 size 134x23; Text 'NIVEL DE AGUA'
   TextField "Campo de texto_32" at 193,240 size 140x23; Text 'AGUA CALIENTE'
   TextField "Campo de texto_34" at 193,304 size 132x23; Text 'TEMPERATURA'
   TextField "Campo de texto_35" at 193,336 size 70x23; Text 'TIEMPO'
   TextField "Campo de texto_36" at 193,368 size 134x23; Text 'NIVEL DE AGUA'
   TextField "Campo de texto_37" at 193,400 size 140x23; Text 'AGUA CALIENTE'
   TextField "Campo de texto_38" at 193,432 size 132x23; Text 'TEMPERATURA'
   TextField "Campo de texto_39" at 193,464 size 70x23; Text 'TIEMPO'
   TextField "Campo de texto_40" at 193,496 size 134x23; Text 'NIVEL DE AGUA'
   TextField "Campo de texto_41" at 193,528 size 140x23; Text 'AGUA CALIENTE'
   TextField "Campo de texto_42" at 193,560 size 132x23; Text 'TEMPERATURA'
   TextField "Campo de texto_43" at 193,592 size 94x23; Text 'CANTIDAD'
   TextField "Campo de texto_44" at 193,624 size 70x23; Text 'TIEMPO'
   TextField "Campo de texto_45" at 193,656 size 70x23; Text 'TIEMPO'
   TextField "Campo de texto_4" at 193,272 size 63x23; Text 'VAPOR'
   TextField "Campo de texto_6" at 193,176 size 70x23; Text 'TIEMPO'
   TextField "Campo de texto_7" at 426,39 size 17x33; Text '9'
   TextField "Campo de texto_8" at 537,39 size 34x33; Text '10'
   TextField "Campo de texto_9" at 657,39 size 34x33; Text '11'
   TextField "Campo de texto_11" at 777,39 size 34x33; Text '12'
   TextField "Campo de texto_12" at 897,39 size 34x33; Text '13'
   TextField "Campo de texto_13" at 1017,39 size 34x33; Text '14'
   TextField "Campo de texto_15" at 1137,39 size 34x33; Text '15'
   TextField "Campo de texto_17" at 778,4 size 159x33; Text 'PROGRAMA'
   Button "Botón_1" at 6,695 size 361x66; TextOff 'ATRAS'
      on Click: ActivateScreen("Prog_Lav3_0", 0)
   Button "Botón_2" at 996,694 size 361x66; TextOff 'SIGUIENTE'
      on Click: ActivateScreen("Prog_Lav4_0", 0)
   Button "Botón_3" at 374,694 size 616x66; TextOff 'PRINCIPAL'
      on Click: ActivateScreen("Principal", 0)
   IOField "Campo ES_1" at 394,656 size 80x24; FormatPattern FF; Unit  M
      ProcessValue <- "Lav3_Prog9_Centr_Tiempo"
   IOField "Campo ES_2" at 394,592 size 80x24; FormatPattern F
      ProcessValue <- "Lav3_Prog9_EnjFin_Cant"
   IOField "Campo ES_3" at 394,624 size 80x24; FormatPattern FF; Unit  M
      ProcessValue <- "Lav3_Prog9_EnjFin_Tiempo"
   IOField "Campo ES_4" at 394,80 size 80x24; FormatPattern F
      ProcessValue <- "Lav3_Prog9_EnjIni_Cant"
   IOField "Campo ES_5" at 394,144 size 80x24; FormatPattern F
      ProcessValue <- "Lav3_Prog9_EnjIni_NivAg"
   IOField "Campo ES_6" at 394,112 size 80x24; FormatPattern FF; Unit  M
      ProcessValue <- "Lav3_Prog9_EnjIni_Tiempo"
   IOField "Campo ES_7" at 394,400 size 80x24; FormatPattern F
      ProcessValue <- "Lav3_Prog9_Lav1_AgCaliente"
   IOField "Campo ES_8" at 394,368 size 80x24; FormatPattern F
      ProcessValue <- "Lav3_Prog9_Lav1_NivAg"
   IOField "Campo ES_9" at 394,432 size 80x24; FormatPattern FF; Unit  °C
      ProcessValue <- "Lav3_Prog9_Lav1_Temperatura"
   IOField "Campo ES_10" at 394,336 size 80x24; FormatPattern FF; Unit  M
      ProcessValue <- "Lav3_Prog9_Lav1_Tiempo"
   IOField "Campo ES_11" at 394,528 size 80x24; FormatPattern F
      ProcessValue <- "Lav3_Prog9_Lav2_AgCaliente"
   IOField "Campo ES_12" at 394,496 size 80x24; FormatPattern F
      ProcessValue <- "Lav3_Prog9_Lav2_NivAg"
   IOField "Campo ES_13" at 394,560 size 80x24; FormatPattern FF; Unit °C
      ProcessValue <- "Lav3_Prog9_Lav2_Temperatura"
   IOField "Campo ES_14" at 394,464 size 80x24; FormatPattern FF; Unit  M
      ProcessValue <- "Lav3_Prog9_Lav2_Tiempo"
   IOField "Campo ES_15" at 394,240 size 80x24; FormatPattern F
      ProcessValue <- "Lav3_Prog9_PreLav_AgCaliente"
   IOField "Campo ES_16" at 394,208 size 80x24; FormatPattern F
      ProcessValue <- "Lav3_Prog9_PreLav_NivAg"
   IOField "Campo ES_17" at 394,304 size 80x24; FormatPattern FF; Unit  °C
      ProcessValue <- "Lav3_Prog9_PreLav_Temperatura"
   IOField "Campo ES_18" at 394,176 size 80x24; FormatPattern FF; Unit  M
      ProcessValue <- "Lav3_Prog9_PreLav_Tiempo"
   IOField "Campo ES_19" at 394,272 size 80x24; FormatPattern F
      ProcessValue <- "Lav3_Prog9_PreLav_Vapor"
   IOField "Campo ES_20" at 514,656 size 80x24; FormatPattern FF; Unit  M
      ProcessValue <- "Lav3_Prog10_Centr_Tiempo"
   IOField "Campo ES_21" at 514,592 size 80x24; FormatPattern F
      ProcessValue <- "Lav3_Prog10_EnjFin_Cant"
   IOField "Campo ES_22" at 514,624 size 80x24; FormatPattern FF; Unit  M
      ProcessValue <- "Lav3_Prog10_EnjFin_Tiempo"
   IOField "Campo ES_23" at 514,80 size 80x24; FormatPattern F
      ProcessValue <- "Lav3_Prog10_EnjIni_Cant"
   IOField "Campo ES_24" at 514,144 size 80x24; FormatPattern F
      ProcessValue <- "Lav3_Prog10_EnjIni_NivAg"
   IOField "Campo ES_25" at 514,112 size 80x24; FormatPattern FF; Unit  M
      ProcessValue <- "Lav3_Prog10_EnjIni_Tiempo"
   IOField "Campo ES_26" at 514,400 size 80x24; FormatPattern F
      ProcessValue <- "Lav3_Prog10_Lav1_AgCaliente"
   IOField "Campo ES_27" at 514,368 size 80x24; FormatPattern F
      ProcessValue <- "Lav3_Prog10_Lav1_NivAg"
   IOField "Campo ES_28" at 514,432 size 80x24; FormatPattern FF; Unit  °C
      ProcessValue <- "Lav3_Prog10_Lav1_Temperatura"
   IOField "Campo ES_29" at 514,336 size 80x24; FormatPattern FF; Unit  M
      ProcessValue <- "Lav3_Prog10_Lav1_Tiempo"
   IOField "Campo ES_30" at 514,528 size 80x24; FormatPattern F
      ProcessValue <- "Lav3_Prog10_Lav2_AgCaliente"
   IOField "Campo ES_31" at 514,496 size 80x24; FormatPattern F
      ProcessValue <- "Lav3_Prog10_Lav2_NivAg"
   IOField "Campo ES_32" at 514,560 size 80x24; FormatPattern FF; Unit °C
      ProcessValue <- "Lav3_Prog10_Lav2_Temperatura"
   IOField "Campo ES_33" at 514,464 size 80x24; FormatPattern FF; Unit  M
      ProcessValue <- "Lav3_Prog10_Lav2_Tiempo"
   IOField "Campo ES_34" at 514,240 size 80x24; FormatPattern F
      ProcessValue <- "Lav3_Prog10_PreLav_AgCaliente"
   IOField "Campo ES_35" at 514,208 size 80x24; FormatPattern F
      ProcessValue <- "Lav3_Prog10_PreLav_NivAg"
   IOField "Campo ES_36" at 514,304 size 80x24; FormatPattern FF; Unit  °C
      ProcessValue <- "Lav3_Prog10_PreLav_Temperatura"
   IOField "Campo ES_37" at 514,176 size 80x24; FormatPattern FF; Unit  M
      ProcessValue <- "Lav3_Prog10_PreLav_Tiempo"
   IOField "Campo ES_38" at 514,272 size 80x24; FormatPattern F
      ProcessValue <- "Lav3_Prog10_PreLav_Vapor"
   IOField "Campo ES_39" at 634,656 size 80x24; FormatPattern FF; Unit  M
      ProcessValue <- "Lav3_Prog11_Centr_Tiempo"
   IOField "Campo ES_40" at 634,592 size 80x24; FormatPattern F
      ProcessValue <- "Lav3_Prog11_EnjFin_Cant"
   IOField "Campo ES_41" at 634,624 size 80x24; FormatPattern FF; Unit  M
      ProcessValue <- "Lav3_Prog11_EnjFin_Tiempo"
   IOField "Campo ES_42" at 634,80 size 80x24; FormatPattern F
      ProcessValue <- "Lav3_Prog11_EnjIni_Cant"
   IOField "Campo ES_43" at 634,144 size 80x24; FormatPattern F
      ProcessValue <- "Lav3_Prog11_EnjIni_NivAg"
   IOField "Campo ES_44" at 634,112 size 80x24; FormatPattern FF; Unit  M
      ProcessValue <- "Lav3_Prog11_EnjIni_Tiempo"
   IOField "Campo ES_45" at 634,400 size 80x24; FormatPattern F
      ProcessValue <- "Lav3_Prog11_Lav1_AgCaliente"
   IOField "Campo ES_46" at 634,368 size 80x24; FormatPattern F
      ProcessValue <- "Lav3_Prog11_Lav1_NivAg"
   IOField "Campo ES_47" at 634,432 size 80x24; FormatPattern FF; Unit  °C
      ProcessValue <- "Lav3_Prog11_Lav1_Temperatura"
   IOField "Campo ES_48" at 634,336 size 80x24; FormatPattern FF; Unit  M
      ProcessValue <- "Lav3_Prog11_Lav1_Tiempo"
   IOField "Campo ES_49" at 634,528 size 80x24; FormatPattern F
      ProcessValue <- "Lav3_Prog11_Lav2_AgCaliente"
   IOField "Campo ES_50" at 634,496 size 80x24; FormatPattern F
      ProcessValue <- "Lav3_Prog11_Lav2_NivAg"
   IOField "Campo ES_51" at 634,560 size 80x24; FormatPattern FF; Unit °C
      ProcessValue <- "Lav3_Prog11_Lav2_Temperatura"
   IOField "Campo ES_52" at 634,464 size 80x24; FormatPattern FF; Unit  M
      ProcessValue <- "Lav3_Prog11_Lav2_Tiempo"
   IOField "Campo ES_53" at 634,240 size 80x24; FormatPattern F
      ProcessValue <- "Lav3_Prog11_PreLav_AgCaliente"
   IOField "Campo ES_54" at 634,208 size 80x24; FormatPattern F
      ProcessValue <- "Lav3_Prog11_PreLav_NivAg"
   IOField "Campo ES_55" at 634,304 size 80x24; FormatPattern FF; Unit  °C
      ProcessValue <- "Lav3_Prog11_PreLav_Temperatura"
   IOField "Campo ES_56" at 634,176 size 80x24; FormatPattern FF; Unit  M
      ProcessValue <- "Lav3_Prog11_PreLav_Tiempo"
   IOField "Campo ES_57" at 634,272 size 80x24; FormatPattern F
      ProcessValue <- "Lav3_Prog11_PreLav_Vapor"
   IOField "Campo ES_58" at 754,656 size 80x24; FormatPattern FF; Unit  M
      ProcessValue <- "Lav3_Prog12_Centr_Tiempo"
   IOField "Campo ES_59" at 754,592 size 80x24; FormatPattern F
      ProcessValue <- "Lav3_Prog12_EnjFin_Cant"
   IOField "Campo ES_60" at 754,624 size 80x24; FormatPattern FF; Unit  M
      ProcessValue <- "Lav3_Prog12_EnjFin_Tiempo"
   IOField "Campo ES_61" at 754,80 size 80x24; FormatPattern F
      ProcessValue <- "Lav3_Prog12_EnjIni_Cant"
   IOField "Campo ES_62" at 754,144 size 80x24; FormatPattern F
      ProcessValue <- "Lav3_Prog12_EnjIni_NivAg"
   IOField "Campo ES_63" at 754,112 size 80x24; FormatPattern FF; Unit  M
      ProcessValue <- "Lav3_Prog12_EnjIni_Tiempo"
   IOField "Campo ES_64" at 754,400 size 80x24; FormatPattern F
      ProcessValue <- "Lav3_Prog12_Lav1_AgCaliente"
   IOField "Campo ES_65" at 754,368 size 80x24; FormatPattern F
      ProcessValue <- "Lav3_Prog12_Lav1_NivAg"
   IOField "Campo ES_66" at 754,432 size 80x24; FormatPattern FF; Unit  °C
      ProcessValue <- "Lav3_Prog12_Lav1_Temperatura"
   IOField "Campo ES_67" at 754,336 size 80x24; FormatPattern FF; Unit  M
      ProcessValue <- "Lav3_Prog12_Lav1_Tiempo"
   IOField "Campo ES_68" at 754,528 size 80x24; FormatPattern F
      ProcessValue <- "Lav3_Prog12_Lav2_AgCaliente"
   IOField "Campo ES_69" at 754,496 size 80x24; FormatPattern F
      ProcessValue <- "Lav3_Prog12_Lav2_NivAg"
   IOField "Campo ES_70" at 754,560 size 80x24; FormatPattern FF; Unit °C
      ProcessValue <- "Lav3_Prog12_Lav2_Temperatura"
   IOField "Campo ES_71" at 754,464 size 80x24; FormatPattern FF; Unit  M
      ProcessValue <- "Lav3_Prog12_Lav2_Tiempo"
   IOField "Campo ES_72" at 754,240 size 80x24; FormatPattern F
      ProcessValue <- "Lav3_Prog12_PreLav_AgCaliente"
   IOField "Campo ES_73" at 754,208 size 80x24; FormatPattern F
      ProcessValue <- "Lav3_Prog12_PreLav_NivAg"
   IOField "Campo ES_74" at 754,304 size 80x24; FormatPattern FF; Unit  °C
      ProcessValue <- "Lav3_Prog12_PreLav_Temperatura"
   IOField "Campo ES_75" at 754,176 size 80x24; FormatPattern FF; Unit  M
      ProcessValue <- "Lav3_Prog12_PreLav_Tiempo"
   IOField "Campo ES_76" at 754,272 size 80x24; FormatPattern F
      ProcessValue <- "Lav3_Prog12_PreLav_Vapor"
   IOField "Campo ES_77" at 874,656 size 80x24; FormatPattern FF; Unit  M
      ProcessValue <- "Lav3_Prog13_Centr_Tiempo"
   IOField "Campo ES_78" at 874,592 size 80x24; FormatPattern F
      ProcessValue <- "Lav3_Prog13_EnjFin_Cant"
   IOField "Campo ES_79" at 874,624 size 80x24; FormatPattern FF; Unit  M
      ProcessValue <- "Lav3_Prog13_EnjFin_Tiempo"
   IOField "Campo ES_80" at 874,80 size 80x24; FormatPattern F
      ProcessValue <- "Lav3_Prog13_EnjIni_Cant"
   IOField "Campo ES_81" at 874,144 size 80x24; FormatPattern F
      ProcessValue <- "Lav3_Prog13_EnjIni_NivAg"
   IOField "Campo ES_82" at 874,112 size 80x24; FormatPattern FF; Unit  M
      ProcessValue <- "Lav3_Prog13_EnjIni_Tiempo"
   IOField "Campo ES_83" at 874,400 size 80x24; FormatPattern F
      ProcessValue <- "Lav3_Prog13_Lav1_AgCaliente"
   IOField "Campo ES_84" at 874,368 size 80x24; FormatPattern F
      ProcessValue <- "Lav3_Prog13_Lav1_NivAg"
   IOField "Campo ES_85" at 874,432 size 80x24; FormatPattern FF; Unit  °C
      ProcessValue <- "Lav3_Prog13_Lav1_Temperatura"
   IOField "Campo ES_86" at 874,336 size 80x24; FormatPattern FF; Unit  M
      ProcessValue <- "Lav3_Prog13_Lav1_Tiempo"
   IOField "Campo ES_87" at 874,528 size 80x24; FormatPattern F
      ProcessValue <- "Lav3_Prog13_Lav2_AgCaliente"
   IOField "Campo ES_88" at 874,496 size 80x24; FormatPattern F
      ProcessValue <- "Lav3_Prog13_Lav2_NivAg"
   IOField "Campo ES_89" at 874,560 size 80x24; FormatPattern FF; Unit °C
      ProcessValue <- "Lav3_Prog13_Lav2_Temperatura"
   IOField "Campo ES_90" at 874,464 size 80x24; FormatPattern FF; Unit  M
      ProcessValue <- "Lav3_Prog13_Lav2_Tiempo"
   IOField "Campo ES_91" at 874,240 size 80x24; FormatPattern F
      ProcessValue <- "Lav3_Prog13_PreLav_AgCaliente"
   IOField "Campo ES_92" at 874,208 size 80x24; FormatPattern F
      ProcessValue <- "Lav3_Prog13_PreLav_NivAg"
   IOField "Campo ES_93" at 874,304 size 80x24; FormatPattern FF; Unit  °C
      ProcessValue <- "Lav3_Prog13_PreLav_Temperatura"
   IOField "Campo ES_94" at 874,176 size 80x24; FormatPattern FF; Unit  M
      ProcessValue <- "Lav3_Prog13_PreLav_Tiempo"
   IOField "Campo ES_95" at 874,272 size 80x24; FormatPattern F
      ProcessValue <- "Lav3_Prog13_PreLav_Vapor"
   IOField "Campo ES_96" at 994,656 size 80x24; FormatPattern FF; Unit  M
      ProcessValue <- "Lav3_Prog14_Centr_Tiempo"
   IOField "Campo ES_97" at 994,592 size 80x24; FormatPattern F
      ProcessValue <- "Lav3_Prog14_EnjFin_Cant"
   IOField "Campo ES_98" at 994,624 size 80x24; FormatPattern FF; Unit  M
      ProcessValue <- "Lav3_Prog14_EnjFin_Tiempo"
   IOField "Campo ES_99" at 994,80 size 80x24; FormatPattern F
      ProcessValue <- "Lav3_Prog14_EnjIni_Cant"
   IOField "Campo ES_100" at 994,144 size 80x24; FormatPattern F
      ProcessValue <- "Lav3_Prog14_EnjIni_NivAg"
   IOField "Campo ES_101" at 994,112 size 80x24; FormatPattern FF; Unit  M
      ProcessValue <- "Lav3_Prog14_EnjIni_Tiempo"
   IOField "Campo ES_102" at 994,400 size 80x24; FormatPattern F
      ProcessValue <- "Lav3_Prog14_Lav1_AgCaliente"
   IOField "Campo ES_103" at 994,368 size 80x24; FormatPattern F
      ProcessValue <- "Lav3_Prog14_Lav1_NivAg"
   IOField "Campo ES_104" at 994,432 size 80x24; FormatPattern FF; Unit  °C
      ProcessValue <- "Lav3_Prog14_Lav1_Temperatura"
   IOField "Campo ES_105" at 994,336 size 80x24; FormatPattern FF; Unit  M
      ProcessValue <- "Lav3_Prog14_Lav1_Tiempo"
   IOField "Campo ES_106" at 994,528 size 80x24; FormatPattern F
      ProcessValue <- "Lav3_Prog14_Lav2_AgCaliente"
   IOField "Campo ES_107" at 994,496 size 80x24; FormatPattern F
      ProcessValue <- "Lav3_Prog14_Lav2_NivAg"
   IOField "Campo ES_108" at 994,560 size 80x24; FormatPattern FF; Unit °C
      ProcessValue <- "Lav3_Prog14_Lav2_Temperatura"
   IOField "Campo ES_109" at 994,464 size 80x24; FormatPattern FF; Unit  M
      ProcessValue <- "Lav3_Prog14_Lav2_Tiempo"
   IOField "Campo ES_110" at 994,240 size 80x24; FormatPattern F
      ProcessValue <- "Lav3_Prog14_PreLav_AgCaliente"
   IOField "Campo ES_111" at 994,208 size 80x24; FormatPattern F
      ProcessValue <- "Lav3_Prog14_PreLav_NivAg"
   IOField "Campo ES_112" at 994,304 size 80x24; FormatPattern FF; Unit  °C
      ProcessValue <- "Lav3_Prog14_PreLav_Temperatura"
   IOField "Campo ES_113" at 994,176 size 80x24; FormatPattern FF; Unit  M
      ProcessValue <- "Lav3_Prog14_PreLav_Tiempo"
   IOField "Campo ES_114" at 994,272 size 80x24; FormatPattern F
      ProcessValue <- "Lav3_Prog14_PreLav_Vapor"
   IOField "Campo ES_115" at 1114,656 size 80x24; FormatPattern FF; Unit  M
      ProcessValue <- "Lav3_Prog15_Centr_Tiempo"
   IOField "Campo ES_116" at 1114,592 size 80x24; FormatPattern F
      ProcessValue <- "Lav3_Prog15_EnjFin_Cant"
   IOField "Campo ES_117" at 1114,624 size 80x24; FormatPattern FF; Unit  M
      ProcessValue <- "Lav3_Prog15_EnjFin_Tiempo"
   IOField "Campo ES_118" at 1114,80 size 80x24; FormatPattern F
      ProcessValue <- "Lav3_Prog15_EnjIni_Cant"
   IOField "Campo ES_119" at 1114,144 size 80x24; FormatPattern F
      ProcessValue <- "Lav3_Prog15_EnjIni_NivAg"
   IOField "Campo ES_120" at 1114,112 size 80x24; FormatPattern FF; Unit  M
      ProcessValue <- "Lav3_Prog15_EnjIni_Tiempo"
   IOField "Campo ES_121" at 1114,400 size 80x24; FormatPattern F
      ProcessValue <- "Lav3_Prog15_Lav1_AgCaliente"
   IOField "Campo ES_122" at 1114,368 size 80x24; FormatPattern F
      ProcessValue <- "Lav3_Prog15_Lav1_NivAg"
   IOField "Campo ES_123" at 1114,432 size 80x24; FormatPattern FF; Unit  °C
      ProcessValue <- "Lav3_Prog15_Lav1_Temperatura"
   IOField "Campo ES_124" at 1114,336 size 80x24; FormatPattern FF; Unit  M
      ProcessValue <- "Lav3_Prog15_Lav1_Tiempo"
   IOField "Campo ES_125" at 1114,528 size 80x24; FormatPattern F
      ProcessValue <- "Lav3_Prog15_Lav2_AgCaliente"
   IOField "Campo ES_126" at 1114,496 size 80x24; FormatPattern F
      ProcessValue <- "Lav3_Prog15_Lav2_NivAg"
   IOField "Campo ES_127" at 1114,560 size 80x24; FormatPattern FF; Unit °C
      ProcessValue <- "Lav3_Prog15_Lav2_Temperatura"
   IOField "Campo ES_128" at 1114,464 size 80x24; FormatPattern FF; Unit  M
      ProcessValue <- "Lav3_Prog15_Lav2_Tiempo"
   IOField "Campo ES_129" at 1114,240 size 80x24; FormatPattern F
      ProcessValue <- "Lav3_Prog15_PreLav_AgCaliente"
   IOField "Campo ES_130" at 1114,208 size 80x24; FormatPattern F
      ProcessValue <- "Lav3_Prog15_PreLav_NivAg"
   IOField "Campo ES_131" at 1114,304 size 80x24; FormatPattern FF; Unit  °C
      ProcessValue <- "Lav3_Prog15_PreLav_Temperatura"
   IOField "Campo ES_132" at 1114,176 size 80x24; FormatPattern FF; Unit  M
      ProcessValue <- "Lav3_Prog15_PreLav_Tiempo"
   IOField "Campo ES_133" at 1114,272 size 80x24; FormatPattern F
      ProcessValue <- "Lav3_Prog15_PreLav_Vapor"

screen "Prog_Lav4_0" 1366x768
   TextField "Campo de texto_1" at 49,16 size 194x39; Text 'LAVADORA 4'
   TextField "Campo de texto_2" at 49,80 size 103x23; Text 'ENJUAGUES'
   TextField "Campo de texto_3" at 49,112 size 90x23; Text 'INICIALES'
   TextField "Campo de texto_5" at 49,176 size 113x23; Text 'PRE-LAVADO'
   TextField "Campo de texto_10" at 49,336 size 88x23; Text 'LAVADO 1'
   TextField "Campo de texto_14" at 49,464 size 88x23; Text 'LAVADO 2'
   TextField "Campo de texto_18" at 49,592 size 103x23; Text 'ENJUAGUES'
   TextField "Campo de texto_19" at 49,624 size 74x23; Text 'FINALES'
   TextField "Campo de texto_20" at 49,656 size 137x23; Text 'CENTRIFUGADO'
   TextField "Campo de texto_27" at 193,80 size 94x23; Text 'CANTIDAD'
   TextField "Campo de texto_28" at 193,144 size 134x23; Text 'NIVEL DE AGUA'
   TextField "Campo de texto_29" at 193,112 size 70x23; Text 'TIEMPO'
   TextField "Campo de texto_30" at 193,208 size 134x23; Text 'NIVEL DE AGUA'
   TextField "Campo de texto_32" at 193,240 size 140x23; Text 'AGUA CALIENTE'
   TextField "Campo de texto_34" at 193,304 size 132x23; Text 'TEMPERATURA'
   TextField "Campo de texto_35" at 193,336 size 70x23; Text 'TIEMPO'
   TextField "Campo de texto_36" at 193,368 size 134x23; Text 'NIVEL DE AGUA'
   TextField "Campo de texto_37" at 193,400 size 140x23; Text 'AGUA CALIENTE'
   TextField "Campo de texto_38" at 193,432 size 132x23; Text 'TEMPERATURA'
   TextField "Campo de texto_39" at 193,464 size 70x23; Text 'TIEMPO'
   TextField "Campo de texto_40" at 193,496 size 134x23; Text 'NIVEL DE AGUA'
   TextField "Campo de texto_41" at 193,528 size 140x23; Text 'AGUA CALIENTE'
   TextField "Campo de texto_42" at 193,560 size 132x23; Text 'TEMPERATURA'
   TextField "Campo de texto_43" at 193,592 size 94x23; Text 'CANTIDAD'
   TextField "Campo de texto_44" at 193,624 size 70x23; Text 'TIEMPO'
   TextField "Campo de texto_45" at 193,656 size 70x23; Text 'TIEMPO'
   TextField "Campo de texto_4" at 193,272 size 63x23; Text 'VAPOR'
   TextField "Campo de texto_6" at 193,176 size 70x23; Text 'TIEMPO'
   TextField "Campo de texto_7" at 426,39 size 17x33; Text '1'
   TextField "Campo de texto_8" at 546,39 size 17x33; Text '2'
   TextField "Campo de texto_9" at 666,39 size 17x33; Text '3'
   TextField "Campo de texto_11" at 786,39 size 17x33; Text '4'
   TextField "Campo de texto_12" at 906,39 size 17x33; Text '5'
   TextField "Campo de texto_13" at 1026,39 size 17x33; Text '6'
   TextField "Campo de texto_15" at 1146,39 size 17x33; Text '7'
   TextField "Campo de texto_16" at 1266,39 size 17x33; Text '8'
   TextField "Campo de texto_17" at 778,4 size 159x33; Text 'PROGRAMA'
   Button "Botón_1" at 6,695 size 361x66; TextOff 'ATRAS'
      on Click: ActivateScreen("Prog_Lav3_1", 0)
   Button "Botón_2" at 996,694 size 361x66; TextOff 'SIGUIENTE'
      on Click: ActivateScreen("Prog_Lav4_1", 0)
   Button "Botón_3" at 374,694 size 616x66; TextOff 'PRINCIPAL'
      on Click: ActivateScreen("Principal", 0)
   IOField "Campo ES_1" at 394,656 size 80x24; FormatPattern FF; Unit  M
      ProcessValue <- "Lav4_Prog1_Centr_Tiempo"
   IOField "Campo ES_2" at 394,592 size 80x24; FormatPattern F
      ProcessValue <- "Lav4_Prog1_EnjFin_Cant"
   IOField "Campo ES_3" at 394,624 size 80x24; FormatPattern FF; Unit  M
      ProcessValue <- "Lav4_Prog1_EnjFin_Tiempo"
   IOField "Campo ES_4" at 394,80 size 80x24; FormatPattern F
      ProcessValue <- "Lav4_Prog1_EnjIni_Cant"
   IOField "Campo ES_5" at 394,144 size 80x24; FormatPattern F
      ProcessValue <- "Lav4_Prog1_EnjIni_NivAg"
   IOField "Campo ES_6" at 394,112 size 80x24; FormatPattern FF; Unit  M
      ProcessValue <- "Lav4_Prog1_EnjIni_Tiempo"
   IOField "Campo ES_7" at 394,400 size 80x24; FormatPattern F
      ProcessValue <- "Lav4_Prog1_Lav1_AgCaliente"
   IOField "Campo ES_8" at 394,368 size 80x24; FormatPattern F
      ProcessValue <- "Lav4_Prog1_Lav1_NivAg"
   IOField "Campo ES_9" at 394,432 size 80x24; FormatPattern FF; Unit  °C
      ProcessValue <- "Lav4_Prog1_Lav1_Temperatura"
   IOField "Campo ES_10" at 394,336 size 80x24; FormatPattern FF; Unit  M
      ProcessValue <- "Lav4_Prog1_Lav1_Tiempo"
   IOField "Campo ES_11" at 394,528 size 80x24; FormatPattern F
      ProcessValue <- "Lav4_Prog1_Lav2_AgCaliente"
   IOField "Campo ES_12" at 394,496 size 80x24; FormatPattern F
      ProcessValue <- "Lav4_Prog1_Lav2_NivAg"
   IOField "Campo ES_13" at 394,560 size 80x24; FormatPattern FF; Unit °C
      ProcessValue <- "Lav4_Prog1_Lav2_Temperatura"
   IOField "Campo ES_14" at 394,464 size 80x24; FormatPattern FF; Unit  M
      ProcessValue <- "Lav4_Prog1_Lav2_Tiempo"
   IOField "Campo ES_15" at 394,240 size 80x24; FormatPattern F
      ProcessValue <- "Lav4_Prog1_PreLav_AgCaliente"
   IOField "Campo ES_16" at 394,208 size 80x24; FormatPattern F
      ProcessValue <- "Lav4_Prog1_PreLav_NivAg"
   IOField "Campo ES_17" at 394,304 size 80x24; FormatPattern FF; Unit  °C
      ProcessValue <- "Lav4_Prog1_PreLav_Temperatura"
   IOField "Campo ES_18" at 394,176 size 80x24; FormatPattern FF; Unit  M
      ProcessValue <- "Lav4_Prog1_PreLav_Tiempo"
   IOField "Campo ES_19" at 394,272 size 80x24; FormatPattern F
      ProcessValue <- "Lav4_Prog1_PreLav_Vapor"
   IOField "Campo ES_20" at 514,656 size 80x24; FormatPattern FF; Unit  M
      ProcessValue <- "Lav4_Prog2_Centr_Tiempo"
   IOField "Campo ES_21" at 514,592 size 80x24; FormatPattern F
      ProcessValue <- "Lav4_Prog2_EnjFin_Cant"
   IOField "Campo ES_22" at 514,624 size 80x24; FormatPattern FF; Unit  M
      ProcessValue <- "Lav4_Prog2_EnjFin_Tiempo"
   IOField "Campo ES_23" at 514,80 size 80x24; FormatPattern F
      ProcessValue <- "Lav4_Prog2_EnjIni_Cant"
   IOField "Campo ES_24" at 514,144 size 80x24; FormatPattern F
      ProcessValue <- "Lav4_Prog2_EnjIni_NivAg"
   IOField "Campo ES_25" at 514,112 size 80x24; FormatPattern FF; Unit  M
      ProcessValue <- "Lav4_Prog2_EnjIni_Tiempo"
   IOField "Campo ES_26" at 514,400 size 80x24; FormatPattern F
      ProcessValue <- "Lav4_Prog2_Lav1_AgCaliente"
   IOField "Campo ES_27" at 514,368 size 80x24; FormatPattern F
      ProcessValue <- "Lav4_Prog2_Lav1_NivAg"
   IOField "Campo ES_28" at 514,432 size 80x24; FormatPattern FF; Unit  °C
      ProcessValue <- "Lav4_Prog2_Lav1_Temperatura"
   IOField "Campo ES_29" at 514,336 size 80x24; FormatPattern FF; Unit  M
      ProcessValue <- "Lav4_Prog2_Lav1_Tiempo"
   IOField "Campo ES_30" at 514,528 size 80x24; FormatPattern F
      ProcessValue <- "Lav4_Prog2_Lav2_AgCaliente"
   IOField "Campo ES_31" at 514,496 size 80x24; FormatPattern F
      ProcessValue <- "Lav4_Prog2_Lav2_NivAg"
   IOField "Campo ES_32" at 514,560 size 80x24; FormatPattern FF; Unit °C
      ProcessValue <- "Lav4_Prog2_Lav2_Temperatura"
   IOField "Campo ES_33" at 514,464 size 80x24; FormatPattern FF; Unit  M
      ProcessValue <- "Lav4_Prog2_Lav2_Tiempo"
   IOField "Campo ES_34" at 514,240 size 80x24; FormatPattern F
      ProcessValue <- "Lav4_Prog2_PreLav_AgCaliente"
   IOField "Campo ES_35" at 514,208 size 80x24; FormatPattern F
      ProcessValue <- "Lav4_Prog2_PreLav_NivAg"
   IOField "Campo ES_36" at 514,304 size 80x24; FormatPattern FF; Unit  °C
      ProcessValue <- "Lav4_Prog2_PreLav_Temperatura"
   IOField "Campo ES_37" at 514,176 size 80x24; FormatPattern FF; Unit  M
      ProcessValue <- "Lav4_Prog2_PreLav_Tiempo"
   IOField "Campo ES_38" at 514,272 size 80x24; FormatPattern F
      ProcessValue <- "Lav4_Prog2_PreLav_Vapor"
   IOField "Campo ES_39" at 634,656 size 80x24; FormatPattern FF; Unit  M
      ProcessValue <- "Lav4_Prog3_Centr_Tiempo"
   IOField "Campo ES_40" at 634,592 size 80x24; FormatPattern F
      ProcessValue <- "Lav4_Prog3_EnjFin_Cant"
   IOField "Campo ES_41" at 634,624 size 80x24; FormatPattern FF; Unit  M
      ProcessValue <- "Lav4_Prog3_EnjFin_Tiempo"
   IOField "Campo ES_42" at 634,80 size 80x24; FormatPattern F
      ProcessValue <- "Lav4_Prog3_EnjIni_Cant"
   IOField "Campo ES_43" at 634,144 size 80x24; FormatPattern F
      ProcessValue <- "Lav4_Prog3_EnjIni_NivAg"
   IOField "Campo ES_44" at 634,112 size 80x24; FormatPattern FF; Unit  M
      ProcessValue <- "Lav4_Prog3_EnjIni_Tiempo"
   IOField "Campo ES_45" at 634,400 size 80x24; FormatPattern F
      ProcessValue <- "Lav4_Prog3_Lav1_AgCaliente"
   IOField "Campo ES_46" at 634,368 size 80x24; FormatPattern F
      ProcessValue <- "Lav4_Prog3_Lav1_NivAg"
   IOField "Campo ES_47" at 634,432 size 80x24; FormatPattern FF; Unit  °C
      ProcessValue <- "Lav4_Prog3_Lav1_Temperatura"
   IOField "Campo ES_48" at 634,336 size 80x24; FormatPattern FF; Unit  M
      ProcessValue <- "Lav4_Prog3_Lav1_Tiempo"
   IOField "Campo ES_49" at 634,528 size 80x24; FormatPattern F
      ProcessValue <- "Lav4_Prog3_Lav2_AgCaliente"
   IOField "Campo ES_50" at 634,496 size 80x24; FormatPattern F
      ProcessValue <- "Lav4_Prog3_Lav2_NivAg"
   IOField "Campo ES_51" at 634,560 size 80x24; FormatPattern FF; Unit °C
      ProcessValue <- "Lav4_Prog3_Lav2_Temperatura"
   IOField "Campo ES_52" at 634,464 size 80x24; FormatPattern FF; Unit  M
      ProcessValue <- "Lav4_Prog3_Lav2_Tiempo"
   IOField "Campo ES_53" at 634,240 size 80x24; FormatPattern F
      ProcessValue <- "Lav4_Prog3_PreLav_AgCaliente"
   IOField "Campo ES_54" at 634,208 size 80x24; FormatPattern F
      ProcessValue <- "Lav4_Prog3_PreLav_NivAg"
   IOField "Campo ES_55" at 634,304 size 80x24; FormatPattern FF; Unit  °C
      ProcessValue <- "Lav4_Prog3_PreLav_Temperatura"
   IOField "Campo ES_56" at 634,176 size 80x24; FormatPattern FF; Unit  M
      ProcessValue <- "Lav4_Prog3_PreLav_Tiempo"
   IOField "Campo ES_57" at 634,272 size 80x24; FormatPattern F
      ProcessValue <- "Lav4_Prog3_PreLav_Vapor"
   IOField "Campo ES_58" at 754,656 size 80x24; FormatPattern FF; Unit  M
      ProcessValue <- "Lav4_Prog4_Centr_Tiempo"
   IOField "Campo ES_59" at 754,592 size 80x24; FormatPattern F
      ProcessValue <- "Lav4_Prog4_EnjFin_Cant"
   IOField "Campo ES_60" at 754,624 size 80x24; FormatPattern FF; Unit  M
      ProcessValue <- "Lav4_Prog4_EnjFin_Tiempo"
   IOField "Campo ES_61" at 754,80 size 80x24; FormatPattern F
      ProcessValue <- "Lav4_Prog4_EnjIni_Cant"
   IOField "Campo ES_62" at 754,144 size 80x24; FormatPattern F
      ProcessValue <- "Lav4_Prog4_EnjIni_NivAg"
   IOField "Campo ES_63" at 754,112 size 80x24; FormatPattern FF; Unit  M
      ProcessValue <- "Lav4_Prog4_EnjIni_Tiempo"
   IOField "Campo ES_64" at 754,400 size 80x24; FormatPattern F
      ProcessValue <- "Lav4_Prog4_Lav1_AgCaliente"
   IOField "Campo ES_65" at 754,368 size 80x24; FormatPattern F
      ProcessValue <- "Lav4_Prog4_Lav1_NivAg"
   IOField "Campo ES_66" at 754,432 size 80x24; FormatPattern FF; Unit  °C
      ProcessValue <- "Lav4_Prog4_Lav1_Temperatura"
   IOField "Campo ES_67" at 754,336 size 80x24; FormatPattern FF; Unit  M
      ProcessValue <- "Lav4_Prog4_Lav1_Tiempo"
   IOField "Campo ES_68" at 754,528 size 80x24; FormatPattern F
      ProcessValue <- "Lav4_Prog4_Lav2_AgCaliente"
   IOField "Campo ES_69" at 754,496 size 80x24; FormatPattern F
      ProcessValue <- "Lav4_Prog4_Lav2_NivAg"
   IOField "Campo ES_70" at 754,560 size 80x24; FormatPattern FF; Unit °C
      ProcessValue <- "Lav4_Prog4_Lav2_Temperatura"
   IOField "Campo ES_71" at 754,464 size 80x24; FormatPattern FF; Unit  M
      ProcessValue <- "Lav4_Prog4_Lav2_Tiempo"
   IOField "Campo ES_72" at 754,240 size 80x24; FormatPattern F
      ProcessValue <- "Lav4_Prog4_PreLav_AgCaliente"
   IOField "Campo ES_73" at 754,208 size 80x24; FormatPattern F
      ProcessValue <- "Lav4_Prog4_PreLav_NivAg"
   IOField "Campo ES_74" at 754,304 size 80x24; FormatPattern FF; Unit  °C
      ProcessValue <- "Lav4_Prog4_PreLav_Temperatura"
   IOField "Campo ES_75" at 754,176 size 80x24; FormatPattern FF; Unit  M
      ProcessValue <- "Lav4_Prog4_PreLav_Tiempo"
   IOField "Campo ES_76" at 754,272 size 80x24; FormatPattern F
      ProcessValue <- "Lav4_Prog4_PreLav_Vapor"
   IOField "Campo ES_77" at 874,656 size 80x24; FormatPattern FF; Unit  M
      ProcessValue <- "Lav4_Prog6_Centr_Tiempo"
   IOField "Campo ES_78" at 874,592 size 80x24; FormatPattern F
      ProcessValue <- "Lav4_Prog6_EnjFin_Cant"
   IOField "Campo ES_79" at 874,624 size 80x24; FormatPattern FF; Unit  M
      ProcessValue <- "Lav4_Prog6_EnjFin_Tiempo"
   IOField "Campo ES_80" at 874,80 size 80x24; FormatPattern F
      ProcessValue <- "Lav4_Prog5_EnjIni_Cant"
   IOField "Campo ES_81" at 874,144 size 80x24; FormatPattern F
      ProcessValue <- "Lav4_Prog5_EnjIni_NivAg"
   IOField "Campo ES_82" at 874,112 size 80x24; FormatPattern FF; Unit  M
      ProcessValue <- "Lav4_Prog5_EnjIni_Tiempo"
   IOField "Campo ES_83" at 874,400 size 80x24; FormatPattern F
      ProcessValue <- "Lav4_Prog5_Lav1_AgCaliente"
   IOField "Campo ES_84" at 874,368 size 80x24; FormatPattern F
      ProcessValue <- "Lav4_Prog5_Lav1_NivAg"
   IOField "Campo ES_85" at 874,432 size 80x24; FormatPattern FF; Unit  °C
      ProcessValue <- "Lav4_Prog5_Lav1_Temperatura"
   IOField "Campo ES_86" at 874,336 size 80x24; FormatPattern FF; Unit  M
      ProcessValue <- "Lav4_Prog5_Lav1_Tiempo"
   IOField "Campo ES_87" at 874,528 size 80x24; FormatPattern F
      ProcessValue <- "Lav4_Prog6_Lav2_AgCaliente"
   IOField "Campo ES_88" at 874,496 size 80x24; FormatPattern F
      ProcessValue <- "Lav4_Prog6_Lav2_NivAg"
   IOField "Campo ES_89" at 874,560 size 80x24; FormatPattern FF; Unit °C
      ProcessValue <- "Lav4_Prog6_Lav2_Temperatura"
   IOField "Campo ES_90" at 874,464 size 80x24; FormatPattern FF; Unit  M
      ProcessValue <- "Lav4_Prog6_Lav2_Tiempo"
   IOField "Campo ES_91" at 874,240 size 80x24; FormatPattern F
      ProcessValue <- "Lav4_Prog5_PreLav_AgCaliente"
   IOField "Campo ES_92" at 874,208 size 80x24; FormatPattern F
      ProcessValue <- "Lav4_Prog5_PreLav_NivAg"
   IOField "Campo ES_93" at 874,304 size 80x24; FormatPattern FF; Unit  °C
      ProcessValue <- "Lav4_Prog5_PreLav_Temperatura"
   IOField "Campo ES_94" at 874,176 size 80x24; FormatPattern FF; Unit  M
      ProcessValue <- "Lav4_Prog5_PreLav_Tiempo"
   IOField "Campo ES_95" at 874,272 size 80x24; FormatPattern F
      ProcessValue <- "Lav4_Prog5_PreLav_Vapor"
   IOField "Campo ES_96" at 994,656 size 80x24; FormatPattern FF; Unit  M
      ProcessValue <- "Lav4_Prog6_Centr_Tiempo"
   IOField "Campo ES_97" at 994,592 size 80x24; FormatPattern F
      ProcessValue <- "Lav4_Prog6_EnjFin_Cant"
   IOField "Campo ES_98" at 994,624 size 80x24; FormatPattern FF; Unit  M
      ProcessValue <- "Lav4_Prog6_EnjFin_Tiempo"
   IOField "Campo ES_99" at 994,80 size 80x24; FormatPattern F
      ProcessValue <- "Lav4_Prog6_EnjIni_Cant"
   IOField "Campo ES_100" at 994,144 size 80x24; FormatPattern F
      ProcessValue <- "Lav4_Prog6_EnjIni_NivAg"
   IOField "Campo ES_101" at 994,112 size 80x24; FormatPattern FF; Unit  M
      ProcessValue <- "Lav4_Prog6_EnjIni_Tiempo"
   IOField "Campo ES_102" at 994,400 size 80x24; FormatPattern F
      ProcessValue <- "Lav4_Prog6_Lav1_AgCaliente"
   IOField "Campo ES_103" at 994,368 size 80x24; FormatPattern F
      ProcessValue <- "Lav4_Prog6_Lav1_NivAg"
   IOField "Campo ES_104" at 994,432 size 80x24; FormatPattern FF; Unit  °C
      ProcessValue <- "Lav4_Prog6_Lav1_Temperatura"
   IOField "Campo ES_105" at 994,336 size 80x24; FormatPattern FF; Unit  M
      ProcessValue <- "Lav4_Prog6_Lav1_Tiempo"
   IOField "Campo ES_106" at 994,528 size 80x24; FormatPattern F
      ProcessValue <- "Lav4_Prog6_Lav2_AgCaliente"
   IOField "Campo ES_107" at 994,496 size 80x24; FormatPattern F
      ProcessValue <- "Lav4_Prog6_Lav2_NivAg"
   IOField "Campo ES_108" at 994,560 size 80x24; FormatPattern FF; Unit °C
      ProcessValue <- "Lav4_Prog6_Lav2_Temperatura"
   IOField "Campo ES_109" at 994,464 size 80x24; FormatPattern FF; Unit  M
      ProcessValue <- "Lav4_Prog6_Lav2_Tiempo"
   IOField "Campo ES_110" at 994,240 size 80x24; FormatPattern F
      ProcessValue <- "Lav4_Prog6_PreLav_AgCaliente"
   IOField "Campo ES_111" at 994,208 size 80x24; FormatPattern F
      ProcessValue <- "Lav4_Prog6_PreLav_NivAg"
   IOField "Campo ES_112" at 994,304 size 80x24; FormatPattern FF; Unit  °C
      ProcessValue <- "Lav4_Prog6_PreLav_Temperatura"
   IOField "Campo ES_113" at 994,176 size 80x24; FormatPattern FF; Unit  M
      ProcessValue <- "Lav4_Prog6_PreLav_Tiempo"
   IOField "Campo ES_114" at 994,272 size 80x24; FormatPattern F
      ProcessValue <- "Lav4_Prog6_PreLav_Vapor"
   IOField "Campo ES_115" at 1114,656 size 80x24; FormatPattern FF; Unit  M
      ProcessValue <- "Lav4_Prog7_Centr_Tiempo"
   IOField "Campo ES_116" at 1114,592 size 80x24; FormatPattern F
      ProcessValue <- "Lav4_Prog7_EnjFin_Cant"
   IOField "Campo ES_117" at 1114,624 size 80x24; FormatPattern FF; Unit  M
      ProcessValue <- "Lav4_Prog7_EnjFin_Tiempo"
   IOField "Campo ES_118" at 1114,80 size 80x24; FormatPattern F
      ProcessValue <- "Lav4_Prog7_EnjIni_Cant"
   IOField "Campo ES_119" at 1114,144 size 80x24; FormatPattern F
      ProcessValue <- "Lav4_Prog7_EnjIni_NivAg"
   IOField "Campo ES_120" at 1114,112 size 80x24; FormatPattern FF; Unit  M
      ProcessValue <- "Lav4_Prog7_EnjIni_Tiempo"
   IOField "Campo ES_121" at 1114,400 size 80x24; FormatPattern F
      ProcessValue <- "Lav4_Prog7_Lav1_AgCaliente"
   IOField "Campo ES_122" at 1114,368 size 80x24; FormatPattern F
      ProcessValue <- "Lav4_Prog7_Lav1_NivAg"
   IOField "Campo ES_123" at 1114,432 size 80x24; FormatPattern FF; Unit  °C
      ProcessValue <- "Lav4_Prog7_Lav1_Temperatura"
   IOField "Campo ES_124" at 1114,336 size 80x24; FormatPattern FF; Unit  M
      ProcessValue <- "Lav4_Prog7_Lav1_Tiempo"
   IOField "Campo ES_125" at 1114,528 size 80x24; FormatPattern F
      ProcessValue <- "Lav4_Prog7_Lav2_AgCaliente"
   IOField "Campo ES_126" at 1114,496 size 80x24; FormatPattern F
      ProcessValue <- "Lav4_Prog7_Lav2_NivAg"
   IOField "Campo ES_127" at 1114,560 size 80x24; FormatPattern FF; Unit °C
      ProcessValue <- "Lav4_Prog7_Lav2_Temperatura"
   IOField "Campo ES_128" at 1114,464 size 80x24; FormatPattern FF; Unit  M
      ProcessValue <- "Lav4_Prog7_Lav2_Tiempo"
   IOField "Campo ES_129" at 1114,240 size 80x24; FormatPattern F
      ProcessValue <- "Lav4_Prog7_PreLav_AgCaliente"
   IOField "Campo ES_130" at 1114,208 size 80x24; FormatPattern F
      ProcessValue <- "Lav4_Prog7_PreLav_NivAg"
   IOField "Campo ES_131" at 1114,304 size 80x24; FormatPattern FF; Unit  °C
      ProcessValue <- "Lav4_Prog7_PreLav_Temperatura"
   IOField "Campo ES_132" at 1114,176 size 80x24; FormatPattern FF; Unit  M
      ProcessValue <- "Lav4_Prog7_PreLav_Tiempo"
   IOField "Campo ES_133" at 1114,272 size 80x24; FormatPattern F
      ProcessValue <- "Lav4_Prog7_PreLav_Vapor"
   IOField "Campo ES_134" at 1234,656 size 80x24; FormatPattern FF; Unit  M
      ProcessValue <- "Lav4_Prog8_Centr_Tiempo"
   IOField "Campo ES_135" at 1234,592 size 80x24; FormatPattern F
      ProcessValue <- "Lav4_Prog8_EnjFin_Cant"
   IOField "Campo ES_136" at 1234,624 size 80x24; FormatPattern FF; Unit  M
      ProcessValue <- "Lav4_Prog8_EnjFin_Tiempo"
   IOField "Campo ES_137" at 1234,80 size 80x24; FormatPattern F
      ProcessValue <- "Lav4_Prog8_EnjIni_Cant"
   IOField "Campo ES_138" at 1234,144 size 80x24; FormatPattern F
      ProcessValue <- "Lav4_Prog8_EnjIni_NivAg"
   IOField "Campo ES_139" at 1234,112 size 80x24; FormatPattern FF; Unit  M
      ProcessValue <- "Lav4_Prog8_EnjIni_Tiempo"
   IOField "Campo ES_140" at 1234,400 size 80x24; FormatPattern F
      ProcessValue <- "Lav4_Prog8_Lav1_AgCaliente"
   IOField "Campo ES_141" at 1234,368 size 80x24; FormatPattern F
      ProcessValue <- "Lav4_Prog8_Lav1_NivAg"
   IOField "Campo ES_142" at 1234,432 size 80x24; FormatPattern FF; Unit  °C
      ProcessValue <- "Lav4_Prog8_Lav1_Temperatura"
   IOField "Campo ES_143" at 1234,336 size 80x24; FormatPattern FF; Unit  M
      ProcessValue <- "Lav4_Prog8_Lav1_Tiempo"
   IOField "Campo ES_144" at 1234,528 size 80x24; FormatPattern F
      ProcessValue <- "Lav4_Prog8_Lav2_AgCaliente"
   IOField "Campo ES_145" at 1234,496 size 80x24; FormatPattern F
      ProcessValue <- "Lav4_Prog8_Lav2_NivAg"
   IOField "Campo ES_146" at 1234,560 size 80x24; FormatPattern FF; Unit °C
      ProcessValue <- "Lav4_Prog8_Lav2_Temperatura"
   IOField "Campo ES_147" at 1234,464 size 80x24; FormatPattern FF; Unit  M
      ProcessValue <- "Lav4_Prog8_Lav2_Tiempo"
   IOField "Campo ES_148" at 1234,240 size 80x24; FormatPattern F
      ProcessValue <- "Lav4_Prog8_PreLav_AgCaliente"
   IOField "Campo ES_149" at 1234,208 size 80x24; FormatPattern F
      ProcessValue <- "Lav4_Prog8_PreLav_NivAg"
   IOField "Campo ES_150" at 1234,304 size 80x24; FormatPattern FF; Unit  °C
      ProcessValue <- "Lav4_Prog8_PreLav_Temperatura"
   IOField "Campo ES_151" at 1234,176 size 80x24; FormatPattern FF; Unit  M
      ProcessValue <- "Lav4_Prog8_PreLav_Tiempo"
   IOField "Campo ES_152" at 1234,272 size 80x24; FormatPattern F
      ProcessValue <- "Lav4_Prog8_PreLav_Vapor"

screen "Prog_Lav4_1" 1366x768
   TextField "Campo de texto_1" at 49,16 size 194x39; Text 'LAVADORA 4'
   TextField "Campo de texto_2" at 49,80 size 103x23; Text 'ENJUAGUES'
   TextField "Campo de texto_3" at 49,112 size 90x23; Text 'INICIALES'
   TextField "Campo de texto_5" at 49,176 size 113x23; Text 'PRE-LAVADO'
   TextField "Campo de texto_10" at 49,336 size 88x23; Text 'LAVADO 1'
   TextField "Campo de texto_14" at 49,464 size 88x23; Text 'LAVADO 2'
   TextField "Campo de texto_18" at 49,592 size 103x23; Text 'ENJUAGUES'
   TextField "Campo de texto_19" at 49,624 size 74x23; Text 'FINALES'
   TextField "Campo de texto_20" at 49,656 size 137x23; Text 'CENTRIFUGADO'
   TextField "Campo de texto_27" at 193,80 size 94x23; Text 'CANTIDAD'
   TextField "Campo de texto_28" at 193,144 size 134x23; Text 'NIVEL DE AGUA'
   TextField "Campo de texto_29" at 193,112 size 70x23; Text 'TIEMPO'
   TextField "Campo de texto_30" at 193,208 size 134x23; Text 'NIVEL DE AGUA'
   TextField "Campo de texto_32" at 193,240 size 140x23; Text 'AGUA CALIENTE'
   TextField "Campo de texto_34" at 193,304 size 132x23; Text 'TEMPERATURA'
   TextField "Campo de texto_35" at 193,336 size 70x23; Text 'TIEMPO'
   TextField "Campo de texto_36" at 193,368 size 134x23; Text 'NIVEL DE AGUA'
   TextField "Campo de texto_37" at 193,400 size 140x23; Text 'AGUA CALIENTE'
   TextField "Campo de texto_38" at 193,432 size 132x23; Text 'TEMPERATURA'
   TextField "Campo de texto_39" at 193,464 size 70x23; Text 'TIEMPO'
   TextField "Campo de texto_40" at 193,496 size 134x23; Text 'NIVEL DE AGUA'
   TextField "Campo de texto_41" at 193,528 size 140x23; Text 'AGUA CALIENTE'
   TextField "Campo de texto_42" at 193,560 size 132x23; Text 'TEMPERATURA'
   TextField "Campo de texto_43" at 193,592 size 94x23; Text 'CANTIDAD'
   TextField "Campo de texto_44" at 193,624 size 70x23; Text 'TIEMPO'
   TextField "Campo de texto_45" at 193,656 size 70x23; Text 'TIEMPO'
   TextField "Campo de texto_4" at 193,272 size 63x23; Text 'VAPOR'
   TextField "Campo de texto_6" at 193,176 size 70x23; Text 'TIEMPO'
   TextField "Campo de texto_7" at 426,39 size 17x33; Text '9'
   TextField "Campo de texto_8" at 537,39 size 34x33; Text '10'
   TextField "Campo de texto_9" at 657,39 size 34x33; Text '11'
   TextField "Campo de texto_11" at 777,39 size 34x33; Text '12'
   TextField "Campo de texto_12" at 897,39 size 34x33; Text '13'
   TextField "Campo de texto_13" at 1017,39 size 34x33; Text '14'
   TextField "Campo de texto_15" at 1137,39 size 34x33; Text '15'
   TextField "Campo de texto_17" at 778,4 size 159x33; Text 'PROGRAMA'
   Button "Botón_1" at 6,695 size 361x66; TextOff 'ATRAS'
      on Click: ActivateScreen("Prog_Lav4_0", 0)
   Button "Botón_3" at 374,694 size 616x66; TextOff 'PRINCIPAL'
      on Click: ActivateScreen("Principal", 0)
   IOField "Campo ES_1" at 394,656 size 80x24; FormatPattern FF; Unit  M
      ProcessValue <- "Lav4_Prog9_Centr_Tiempo"
   IOField "Campo ES_2" at 394,592 size 80x24; FormatPattern F
      ProcessValue <- "Lav4_Prog9_EnjFin_Cant"
   IOField "Campo ES_3" at 394,624 size 80x24; FormatPattern FF; Unit  M
      ProcessValue <- "Lav4_Prog9_EnjFin_Tiempo"
   IOField "Campo ES_4" at 394,80 size 80x24; FormatPattern F
      ProcessValue <- "Lav4_Prog9_EnjIni_Cant"
   IOField "Campo ES_5" at 394,144 size 80x24; FormatPattern F
      ProcessValue <- "Lav4_Prog9_EnjIni_NivAg"
   IOField "Campo ES_6" at 394,112 size 80x24; FormatPattern FF; Unit  M
      ProcessValue <- "Lav4_Prog9_EnjIni_Tiempo"
   IOField "Campo ES_7" at 394,400 size 80x24; FormatPattern F
      ProcessValue <- "Lav4_Prog9_Lav1_AgCaliente"
   IOField "Campo ES_8" at 394,368 size 80x24; FormatPattern F
      ProcessValue <- "Lav4_Prog9_Lav1_NivAg"
   IOField "Campo ES_9" at 394,432 size 80x24; FormatPattern FF; Unit  °C
      ProcessValue <- "Lav4_Prog9_Lav1_Temperatura"
   IOField "Campo ES_10" at 394,336 size 80x24; FormatPattern FF; Unit  M
      ProcessValue <- "Lav4_Prog9_Lav1_Tiempo"
   IOField "Campo ES_11" at 394,528 size 80x24; FormatPattern F
      ProcessValue <- "Lav4_Prog9_Lav2_AgCaliente"
   IOField "Campo ES_12" at 394,496 size 80x24; FormatPattern F
      ProcessValue <- "Lav4_Prog9_Lav2_NivAg"
   IOField "Campo ES_13" at 394,560 size 80x24; FormatPattern FF; Unit °C
      ProcessValue <- "Lav4_Prog9_Lav2_Temperatura"
   IOField "Campo ES_14" at 394,464 size 80x24; FormatPattern FF; Unit  M
      ProcessValue <- "Lav4_Prog9_Lav2_Tiempo"
   IOField "Campo ES_15" at 394,240 size 80x24; FormatPattern F
      ProcessValue <- "Lav4_Prog9_PreLav_AgCaliente"
   IOField "Campo ES_16" at 394,208 size 80x24; FormatPattern F
      ProcessValue <- "Lav4_Prog9_PreLav_NivAg"
   IOField "Campo ES_17" at 394,304 size 80x24; FormatPattern FF; Unit  °C
      ProcessValue <- "Lav4_Prog9_PreLav_Temperatura"
   IOField "Campo ES_18" at 394,176 size 80x24; FormatPattern FF; Unit  M
      ProcessValue <- "Lav4_Prog9_PreLav_Tiempo"
   IOField "Campo ES_19" at 394,272 size 80x24; FormatPattern F
      ProcessValue <- "Lav4_Prog9_PreLav_Vapor"
   IOField "Campo ES_20" at 514,656 size 80x24; FormatPattern FF; Unit  M
      ProcessValue <- "Lav4_Prog10_Centr_Tiempo"
   IOField "Campo ES_21" at 514,592 size 80x24; FormatPattern F
      ProcessValue <- "Lav4_Prog10_EnjFin_Cant"
   IOField "Campo ES_22" at 514,624 size 80x24; FormatPattern FF; Unit  M
      ProcessValue <- "Lav4_Prog10_EnjFin_Tiempo"
   IOField "Campo ES_23" at 514,80 size 80x24; FormatPattern F
      ProcessValue <- "Lav4_Prog10_EnjIni_Cant"
   IOField "Campo ES_24" at 514,144 size 80x24; FormatPattern F
      ProcessValue <- "Lav4_Prog10_EnjIni_NivAg"
   IOField "Campo ES_25" at 514,112 size 80x24; FormatPattern FF; Unit  M
      ProcessValue <- "Lav4_Prog10_EnjIni_Tiempo"
   IOField "Campo ES_26" at 514,400 size 80x24; FormatPattern F
      ProcessValue <- "Lav4_Prog10_Lav1_AgCaliente"
   IOField "Campo ES_27" at 514,368 size 80x24; FormatPattern F
      ProcessValue <- "Lav4_Prog10_Lav1_NivAg"
   IOField "Campo ES_28" at 514,432 size 80x24; FormatPattern FF; Unit  °C
      ProcessValue <- "Lav4_Prog10_Lav1_Temperatura"
   IOField "Campo ES_29" at 514,336 size 80x24; FormatPattern FF; Unit  M
      ProcessValue <- "Lav4_Prog10_Lav1_Tiempo"
   IOField "Campo ES_30" at 514,528 size 80x24; FormatPattern F
      ProcessValue <- "Lav4_Prog10_Lav2_AgCaliente"
   IOField "Campo ES_31" at 514,496 size 80x24; FormatPattern F
      ProcessValue <- "Lav4_Prog10_Lav2_NivAg"
   IOField "Campo ES_32" at 514,560 size 80x24; FormatPattern FF; Unit °C
      ProcessValue <- "Lav4_Prog10_Lav2_Temperatura"
   IOField "Campo ES_33" at 514,464 size 80x24; FormatPattern FF; Unit  M
      ProcessValue <- "Lav4_Prog10_Lav2_Tiempo"
   IOField "Campo ES_34" at 514,240 size 80x24; FormatPattern F
      ProcessValue <- "Lav4_Prog10_PreLav_AgCaliente"
   IOField "Campo ES_35" at 514,208 size 80x24; FormatPattern F
      ProcessValue <- "Lav4_Prog10_PreLav_NivAg"
   IOField "Campo ES_36" at 514,304 size 80x24; FormatPattern FF; Unit  °C
      ProcessValue <- "Lav4_Prog10_PreLav_Temperatura"
   IOField "Campo ES_37" at 514,176 size 80x24; FormatPattern FF; Unit  M
      ProcessValue <- "Lav4_Prog10_PreLav_Tiempo"
   IOField "Campo ES_38" at 514,272 size 80x24; FormatPattern F
      ProcessValue <- "Lav4_Prog10_PreLav_Vapor"
   IOField "Campo ES_39" at 634,656 size 80x24; FormatPattern FF; Unit  M
      ProcessValue <- "Lav4_Prog11_Centr_Tiempo"
   IOField "Campo ES_40" at 634,592 size 80x24; FormatPattern F
      ProcessValue <- "Lav4_Prog11_EnjFin_Cant"
   IOField "Campo ES_41" at 634,624 size 80x24; FormatPattern FF; Unit  M
      ProcessValue <- "Lav4_Prog11_EnjFin_Tiempo"
   IOField "Campo ES_42" at 634,80 size 80x24; FormatPattern F
      ProcessValue <- "Lav4_Prog11_EnjIni_Cant"
   IOField "Campo ES_43" at 634,144 size 80x24; FormatPattern F
      ProcessValue <- "Lav4_Prog11_EnjIni_NivAg"
   IOField "Campo ES_44" at 634,112 size 80x24; FormatPattern FF; Unit  M
      ProcessValue <- "Lav4_Prog11_EnjIni_Tiempo"
   IOField "Campo ES_45" at 634,400 size 80x24; FormatPattern F
      ProcessValue <- "Lav4_Prog11_Lav1_AgCaliente"
   IOField "Campo ES_46" at 634,368 size 80x24; FormatPattern F
      ProcessValue <- "Lav4_Prog11_Lav1_NivAg"
   IOField "Campo ES_47" at 634,432 size 80x24; FormatPattern FF; Unit  °C
      ProcessValue <- "Lav4_Prog11_Lav1_Temperatura"
   IOField "Campo ES_48" at 634,336 size 80x24; FormatPattern FF; Unit  M
      ProcessValue <- "Lav4_Prog11_Lav1_Tiempo"
   IOField "Campo ES_49" at 634,528 size 80x24; FormatPattern F
      ProcessValue <- "Lav4_Prog11_Lav2_AgCaliente"
   IOField "Campo ES_50" at 634,496 size 80x24; FormatPattern F
      ProcessValue <- "Lav4_Prog11_Lav2_NivAg"
   IOField "Campo ES_51" at 634,560 size 80x24; FormatPattern FF; Unit °C
      ProcessValue <- "Lav4_Prog11_Lav2_Temperatura"
   IOField "Campo ES_52" at 634,464 size 80x24; FormatPattern FF; Unit  M
      ProcessValue <- "Lav4_Prog11_Lav2_Tiempo"
   IOField "Campo ES_53" at 634,240 size 80x24; FormatPattern F
      ProcessValue <- "Lav4_Prog11_PreLav_AgCaliente"
   IOField "Campo ES_54" at 634,208 size 80x24; FormatPattern F
      ProcessValue <- "Lav4_Prog11_PreLav_NivAg"
   IOField "Campo ES_55" at 634,304 size 80x24; FormatPattern FF; Unit  °C
      ProcessValue <- "Lav4_Prog11_PreLav_Temperatura"
   IOField "Campo ES_56" at 634,176 size 80x24; FormatPattern FF; Unit  M
      ProcessValue <- "Lav4_Prog11_PreLav_Tiempo"
   IOField "Campo ES_57" at 634,272 size 80x24; FormatPattern F
      ProcessValue <- "Lav4_Prog11_PreLav_Vapor"
   IOField "Campo ES_58" at 754,656 size 80x24; FormatPattern FF; Unit  M
      ProcessValue <- "Lav4_Prog12_Centr_Tiempo"
   IOField "Campo ES_59" at 754,592 size 80x24; FormatPattern F
      ProcessValue <- "Lav4_Prog12_EnjFin_Cant"
   IOField "Campo ES_60" at 754,624 size 80x24; FormatPattern FF; Unit  M
      ProcessValue <- "Lav4_Prog12_EnjFin_Tiempo"
   IOField "Campo ES_61" at 754,80 size 80x24; FormatPattern F
      ProcessValue <- "Lav4_Prog12_EnjIni_Cant"
   IOField "Campo ES_62" at 754,144 size 80x24; FormatPattern F
      ProcessValue <- "Lav4_Prog12_EnjIni_NivAg"
   IOField "Campo ES_63" at 754,112 size 80x24; FormatPattern FF; Unit  M
      ProcessValue <- "Lav4_Prog12_EnjIni_Tiempo"
   IOField "Campo ES_64" at 754,400 size 80x24; FormatPattern F
      ProcessValue <- "Lav4_Prog12_Lav1_AgCaliente"
   IOField "Campo ES_65" at 754,368 size 80x24; FormatPattern F
      ProcessValue <- "Lav4_Prog12_Lav1_NivAg"
   IOField "Campo ES_66" at 754,432 size 80x24; FormatPattern FF; Unit  °C
      ProcessValue <- "Lav4_Prog12_Lav1_Temperatura"
   IOField "Campo ES_67" at 754,336 size 80x24; FormatPattern FF; Unit  M
      ProcessValue <- "Lav4_Prog12_Lav1_Tiempo"
   IOField "Campo ES_68" at 754,528 size 80x24; FormatPattern F
      ProcessValue <- "Lav4_Prog12_Lav2_AgCaliente"
   IOField "Campo ES_69" at 754,496 size 80x24; FormatPattern F
      ProcessValue <- "Lav4_Prog12_Lav2_NivAg"
   IOField "Campo ES_70" at 754,560 size 80x24; FormatPattern FF; Unit °C
      ProcessValue <- "Lav4_Prog12_Lav2_Temperatura"
   IOField "Campo ES_71" at 754,464 size 80x24; FormatPattern FF; Unit  M
      ProcessValue <- "Lav4_Prog12_Lav2_Tiempo"
   IOField "Campo ES_72" at 754,240 size 80x24; FormatPattern F
      ProcessValue <- "Lav4_Prog12_PreLav_AgCaliente"
   IOField "Campo ES_73" at 754,208 size 80x24; FormatPattern F
      ProcessValue <- "Lav4_Prog12_PreLav_NivAg"
   IOField "Campo ES_74" at 754,304 size 80x24; FormatPattern FF; Unit  °C
      ProcessValue <- "Lav4_Prog12_PreLav_Temperatura"
   IOField "Campo ES_75" at 754,176 size 80x24; FormatPattern FF; Unit  M
      ProcessValue <- "Lav4_Prog12_PreLav_Tiempo"
   IOField "Campo ES_76" at 754,272 size 80x24; FormatPattern F
      ProcessValue <- "Lav4_Prog12_PreLav_Vapor"
   IOField "Campo ES_77" at 874,656 size 80x24; FormatPattern FF; Unit  M
      ProcessValue <- "Lav4_Prog13_Centr_Tiempo"
   IOField "Campo ES_78" at 874,592 size 80x24; FormatPattern F
      ProcessValue <- "Lav4_Prog13_EnjFin_Cant"
   IOField "Campo ES_79" at 874,624 size 80x24; FormatPattern FF; Unit  M
      ProcessValue <- "Lav4_Prog13_EnjFin_Tiempo"
   IOField "Campo ES_80" at 874,80 size 80x24; FormatPattern F
      ProcessValue <- "Lav4_Prog13_EnjIni_Cant"
   IOField "Campo ES_81" at 874,144 size 80x24; FormatPattern F
      ProcessValue <- "Lav4_Prog13_EnjIni_NivAg"
   IOField "Campo ES_82" at 874,112 size 80x24; FormatPattern FF; Unit  M
      ProcessValue <- "Lav4_Prog13_EnjIni_Tiempo"
   IOField "Campo ES_83" at 874,400 size 80x24; FormatPattern F
      ProcessValue <- "Lav4_Prog13_Lav1_AgCaliente"
   IOField "Campo ES_84" at 874,368 size 80x24; FormatPattern F
      ProcessValue <- "Lav4_Prog13_Lav1_NivAg"
   IOField "Campo ES_85" at 874,432 size 80x24; FormatPattern FF; Unit  °C
      ProcessValue <- "Lav4_Prog13_Lav1_Temperatura"
   IOField "Campo ES_86" at 874,336 size 80x24; FormatPattern FF; Unit  M
      ProcessValue <- "Lav4_Prog13_Lav1_Tiempo"
   IOField "Campo ES_87" at 874,528 size 80x24; FormatPattern F
      ProcessValue <- "Lav4_Prog13_Lav2_AgCaliente"
   IOField "Campo ES_88" at 874,496 size 80x24; FormatPattern F
      ProcessValue <- "Lav4_Prog13_Lav2_NivAg"
   IOField "Campo ES_89" at 874,560 size 80x24; FormatPattern FF; Unit °C
      ProcessValue <- "Lav4_Prog13_Lav2_Temperatura"
   IOField "Campo ES_90" at 874,464 size 80x24; FormatPattern FF; Unit  M
      ProcessValue <- "Lav4_Prog13_Lav2_Tiempo"
   IOField "Campo ES_91" at 874,240 size 80x24; FormatPattern F
      ProcessValue <- "Lav4_Prog13_PreLav_AgCaliente"
   IOField "Campo ES_92" at 874,208 size 80x24; FormatPattern F
      ProcessValue <- "Lav4_Prog13_PreLav_NivAg"
   IOField "Campo ES_93" at 874,304 size 80x24; FormatPattern FF; Unit  °C
      ProcessValue <- "Lav4_Prog13_PreLav_Temperatura"
   IOField "Campo ES_94" at 874,176 size 80x24; FormatPattern FF; Unit  M
      ProcessValue <- "Lav4_Prog13_PreLav_Tiempo"
   IOField "Campo ES_95" at 874,272 size 80x24; FormatPattern F
      ProcessValue <- "Lav4_Prog13_PreLav_Vapor"
   IOField "Campo ES_96" at 994,656 size 80x24; FormatPattern FF; Unit  M
      ProcessValue <- "Lav4_Prog14_Centr_Tiempo"
   IOField "Campo ES_97" at 994,592 size 80x24; FormatPattern F
      ProcessValue <- "Lav4_Prog14_EnjFin_Cant"
   IOField "Campo ES_98" at 994,624 size 80x24; FormatPattern FF; Unit  M
      ProcessValue <- "Lav4_Prog14_EnjFin_Tiempo"
   IOField "Campo ES_99" at 994,80 size 80x24; FormatPattern F
      ProcessValue <- "Lav4_Prog14_EnjIni_Cant"
   IOField "Campo ES_100" at 994,144 size 80x24; FormatPattern F
      ProcessValue <- "Lav4_Prog14_EnjIni_NivAg"
   IOField "Campo ES_101" at 994,112 size 80x24; FormatPattern FF; Unit  M
      ProcessValue <- "Lav4_Prog14_EnjIni_Tiempo"
   IOField "Campo ES_102" at 994,400 size 80x24; FormatPattern F
      ProcessValue <- "Lav4_Prog14_Lav1_AgCaliente"
   IOField "Campo ES_103" at 994,368 size 80x24; FormatPattern F
      ProcessValue <- "Lav4_Prog14_Lav1_NivAg"
   IOField "Campo ES_104" at 994,432 size 80x24; FormatPattern FF; Unit  °C
      ProcessValue <- "Lav4_Prog14_Lav1_Temperatura"
   IOField "Campo ES_105" at 994,336 size 80x24; FormatPattern FF; Unit  M
      ProcessValue <- "Lav4_Prog14_Lav1_Tiempo"
   IOField "Campo ES_106" at 994,528 size 80x24; FormatPattern F
      ProcessValue <- "Lav4_Prog14_Lav2_AgCaliente"
   IOField "Campo ES_107" at 994,496 size 80x24; FormatPattern F
      ProcessValue <- "Lav4_Prog14_Lav2_NivAg"
   IOField "Campo ES_108" at 994,560 size 80x24; FormatPattern FF; Unit °C
      ProcessValue <- "Lav4_Prog14_Lav2_Temperatura"
   IOField "Campo ES_109" at 994,464 size 80x24; FormatPattern FF; Unit  M
      ProcessValue <- "Lav4_Prog14_Lav2_Tiempo"
   IOField "Campo ES_110" at 994,240 size 80x24; FormatPattern F
      ProcessValue <- "Lav4_Prog14_PreLav_AgCaliente"
   IOField "Campo ES_111" at 994,208 size 80x24; FormatPattern F
      ProcessValue <- "Lav4_Prog14_PreLav_NivAg"
   IOField "Campo ES_112" at 994,304 size 80x24; FormatPattern FF; Unit  °C
      ProcessValue <- "Lav4_Prog14_PreLav_Temperatura"
   IOField "Campo ES_113" at 994,176 size 80x24; FormatPattern FF; Unit  M
      ProcessValue <- "Lav4_Prog14_PreLav_Tiempo"
   IOField "Campo ES_114" at 994,272 size 80x24; FormatPattern F
      ProcessValue <- "Lav4_Prog14_PreLav_Vapor"
   IOField "Campo ES_115" at 1114,656 size 80x24; FormatPattern FF; Unit  M
      ProcessValue <- "Lav4_Prog15_Centr_Tiempo"
   IOField "Campo ES_116" at 1114,592 size 80x24; FormatPattern F
      ProcessValue <- "Lav4_Prog15_EnjFin_Cant"
   IOField "Campo ES_117" at 1114,624 size 80x24; FormatPattern FF; Unit  M
      ProcessValue <- "Lav4_Prog15_EnjFin_Tiempo"
   IOField "Campo ES_118" at 1114,80 size 80x24; FormatPattern F
      ProcessValue <- "Lav4_Prog15_EnjIni_Cant"
   IOField "Campo ES_119" at 1114,144 size 80x24; FormatPattern F
      ProcessValue <- "Lav4_Prog15_EnjIni_NivAg"
   IOField "Campo ES_120" at 1114,112 size 80x24; FormatPattern FF; Unit  M
      ProcessValue <- "Lav4_Prog15_EnjIni_Tiempo"
   IOField "Campo ES_121" at 1114,400 size 80x24; FormatPattern F
      ProcessValue <- "Lav4_Prog15_Lav1_AgCaliente"
   IOField "Campo ES_122" at 1114,368 size 80x24; FormatPattern F
      ProcessValue <- "Lav4_Prog15_Lav1_NivAg"
   IOField "Campo ES_123" at 1114,432 size 80x24; FormatPattern FF; Unit  °C
      ProcessValue <- "Lav4_Prog15_Lav1_Temperatura"
   IOField "Campo ES_124" at 1114,336 size 80x24; FormatPattern FF; Unit  M
      ProcessValue <- "Lav4_Prog15_Lav1_Tiempo"
   IOField "Campo ES_125" at 1114,528 size 80x24; FormatPattern F
      ProcessValue <- "Lav4_Prog15_Lav2_AgCaliente"
   IOField "Campo ES_126" at 1114,496 size 80x24; FormatPattern F
      ProcessValue <- "Lav4_Prog15_Lav2_NivAg"
   IOField "Campo ES_127" at 1114,560 size 80x24; FormatPattern FF; Unit °C
      ProcessValue <- "Lav4_Prog15_Lav2_Temperatura"
   IOField "Campo ES_128" at 1114,464 size 80x24; FormatPattern FF; Unit  M
      ProcessValue <- "Lav4_Prog15_Lav2_Tiempo"
   IOField "Campo ES_129" at 1114,240 size 80x24; FormatPattern F
      ProcessValue <- "Lav4_Prog15_PreLav_AgCaliente"
   IOField "Campo ES_130" at 1114,208 size 80x24; FormatPattern F
      ProcessValue <- "Lav4_Prog15_PreLav_NivAg"
   IOField "Campo ES_131" at 1114,304 size 80x24; FormatPattern FF; Unit  °C
      ProcessValue <- "Lav4_Prog15_PreLav_Temperatura"
   IOField "Campo ES_132" at 1114,176 size 80x24; FormatPattern FF; Unit  M
      ProcessValue <- "Lav4_Prog15_PreLav_Tiempo"
   IOField "Campo ES_133" at 1114,272 size 80x24; FormatPattern F
      ProcessValue <- "Lav4_Prog15_PreLav_Vapor"

